//     Term 63 (AT2002-0250)/CC Outputs/Current setpoint value Ch.14 <-> Data Pointer/CurrentSetpointValues[13]
//     Term 63 (AT2002-0250)/CC Outputs/Current setpoint value Ch.15 <-> Data Pointer/CurrentSetpointValues[14]
//     Term 63 (AT2002-0250)/CC Outputs/Current setpoint value Ch.2 <-> Data Pointer/CurrentSetpointValues[1]
//     Term 63 (AT2002-0250)/CC Outputs/Current setpoint value Ch.3 <-> Data Pointer/CurrentSetpointValues[2]
//     Term 63 (AT2002-0250)/CC Outputs/Current setpoint value Ch.4 <-> Data Pointer/CurrentSetpointValues[3]
//     Term 63 (AT2002-0250)/CC Outputs/Current setpoint value Ch.5 <-> Data Pointer/CurrentSetpointValues[4]
//     Term 63 (AT2002-0250)/CC Outputs/Current setpoint value Ch.6 <-> Data Pointer/CurrentSetpointValues[5]
//     Term 63 (AT2002-0250)/CC Outputs/Current setpoint value Ch.7 <-> Data Pointer/CurrentSetpointValues[6]
//     Term 63 (AT2002-0250)/CC Outputs/Current setpoint value Ch.8 <-> Data Pointer/CurrentSetpointValues[7]
//     Term 63 (AT2002-0250)/CC Outputs/Current setpoint value Ch.9 <-> Data Pointer/CurrentSetpointValues[8]
//     Term 63 (AT2002-0250)/Term 64 (AT2002-5250)/FB Inputs/Value Channel 01 <-> Data Pointer/RawPositionValues[0]
//     Term 63 (AT2002-0250)/Term 64 (AT2002-5250)/FB Inputs/Value Channel 02 <-> Data Pointer/RawPositionValues[1]
//     Term 63 (AT2002-0250)/Term 64 (AT2002-5250)/FB Inputs/Value Channel 03 <-> Data Pointer/RawPositionValues[2]
//     Term 63 (AT2002-0250)/Term 64 (AT2002-5250)/FB Inputs/Value Channel 04 <-> Data Pointer/RawPositionValues[3]
//     Term 63 (AT2002-0250)/Term 64 (AT2002-5250)/FB Inputs/Value Channel 05 <-> Data Pointer/RawPositionValues[4]
//     Term 63 (AT2002-0250)/Term 64 (AT2002-5250)/FB Inputs/Value Channel 06 <-> Data Pointer/RawPositionValues[5]
//     Term 63 (AT2002-0250)/Term 64 (AT2002-5250)/FB Inputs/Value Channel 07 <-> Data Pointer/RawPositionValues[6]
//     Term 63 (AT2002-0250)/Term 64 (AT2002-5250)/FB Inputs/Value Channel 08 <-> Data Pointer/RawPositionValues[7]
//     Term 63 (AT2002-0250)/Term 64 (AT2002-5250)/FB Inputs/Value Channel 09 <-> Data Pointer/RawPositionValues[8]
//     Term 63 (AT2002-0250)/Term 64 (AT2002-5250)/FB Inputs/Value Channel 10 <-> Data Pointer/RawPositionValues[9]
//     Term 63 (AT2002-0250)/Term 64 (AT2002-5250)/FB Inputs/Value Channel 11 <-> Data Pointer/RawPositionValues[10]
//     Term 63 (AT2002-0250)/Term 64 (AT2002-5250)/FB Inputs/Value Channel 12 <-> Data Pointer/RawPositionValues[11]
//     Term 63 (AT2002-0250)/Term 64 (AT2002-5250)/FB Inputs/Value Channel 13 <-> Data Pointer/RawPositionValues[12]
//     Term 63 (AT2002-0250)/Term 64 (AT2002-5250)/FB Inputs/Value Channel 14 <-> Data Pointer/RawPositionValues[13]
//     Term 63 (AT2002-0250)/Term 64 (AT2002-5250)/FB Inputs/Value Channel 15 <-> Data Pointer/RawPositionValues[14]
//     Term 63 (AT2002-0250)/Term 64 (AT2002-5250)/FB Inputs/Value Channel 16 <-> Data Pointer/RawPositionValues[15]
//     Term 63 (AT2002-0250)/Term 64 (AT2002-5250)/FB Inputs/Value Channel 17 <-> Data Pointer/RawPositionValues[16]
//     Term 63 (AT2002-0250)/Term 64 (AT2002-5250)/FB Inputs/Value Channel 18 <-> Data Pointer/RawPositionValues[17]
//     Term 63 (AT2002-0250)/Term 64 (AT2002-5250)/FB Inputs/Value Channel 19 <-> Data Pointer/RawPositionValues[18]
//     Term 63 (AT2002-0250)/Term 64 (AT2002-5250)/FB Inputs/Value Channel 20 <-> Data Pointer/RawPositionValues[19]
//     Term 63 (AT2002-0250)/Term 64 (AT2002-5250)/FB Inputs/Value Channel 21 <-> Data Pointer/RawPositionValues[20]
//     Term 63 (AT2002-0250)/Term 64 (AT2002-5250)/FB Inputs/Value Channel 22 <-> Data Pointer/RawPositionValues[21]
//     Term 63 (AT2002-0250)/Term 64 (AT2002-5250)/FB Inputs/Value Channel 23 <-> Data Pointer/RawPositionValues[22]
//     Term 63 (AT2002-0250)/Term 64 (AT2002-5250)/FB Inputs/Value Channel 24 <-> Data Pointer/RawPositionValues[23]
//     Term 63 (AT2002-0250)/Term 64 (AT2002-5250)/FB Inputs/Value Channel 25 <-> Data Pointer/RawPositionValues[24]
//     Term 63 (AT2002-0250)/Term 64 (AT2002-5250)/FB Inputs/Value Channel 26 <-> Data Pointer/RawPositionValues[25]
//     Term 63 (AT2002-0250)/Term 64 (AT2002-5250)/FB Inputs/Value Channel 27 <-> Data Pointer/RawPositionValues[26]
//     Term 63 (AT2002-0250)/Term 64 (AT2002-5250)/FB Inputs/Value Channel 28 <-> Data Pointer/RawPositionValues[27]
//     Term 63 (AT2002-0250)/Term 64 (AT2002-5250)/FB Inputs/Value Channel 29 <-> Data Pointer/RawPositionValues[28]
//     Term 63 (AT2002-0250)/Term 64 (AT2002-5250)/FB Inputs/Value Channel 30 <-> Data Pointer/RawPositionValues[29]
//     Term 63 (AT2002-0250)/Term 64 (AT2002-5250)/FB Inputs/Value Channel 31 <-> Data Pointer/RawPositionValues[30]
//     Term 63 (AT2002-0250)/Term 64 (AT2002-5250)/FB Inputs/Value Channel 32 <-> Data Pointer/RawPositionValues[31]
//   Device 9 <-> TcCOM Objects/XTS ProcessingUnit 1/Part 1/Module 33
//     Term 65 (AT2000-0250)/CC Inputs/Current actual value Ch.1 <-> Data Pointer/CurrentActualValues[0]
//     Term 65 (AT2000-0250)/CC Inputs/Current actual value Ch.10 <-> Data Pointer/CurrentActualValues[9]
//     Term 65 (AT2000-0250)/CC Inputs/Current actual value Ch.11 <-> Data Pointer/CurrentActualValues[10]
//     Term 65 (AT2000-0250)/CC Inputs/Current actual value Ch.12 <-> Data Pointer/CurrentActualValues[11]
//     Term 65 (AT2000-0250)/CC Inputs/Current actual value Ch.13 <-> Data Pointer/CurrentActualValues[12]
//     Term 65 (AT2000-0250)/CC Inputs/Current actual value Ch.14 <-> Data Pointer/CurrentActualValues[13]
//     Term 65 (AT2000-0250)/CC Inputs/Current actual value Ch.15 <-> Data Pointer/CurrentActualValues[14]
//     Term 65 (AT2000-0250)/CC Inputs/Current actual value Ch.2 <-> Data Pointer/CurrentActualValues[1]
//     Term 65 (AT2000-0250)/CC Inputs/Current actual value Ch.3 <-> Data Pointer/CurrentActualValues[2]
//     Term 65 (AT2000-0250)/CC Inputs/Current actual value Ch.4 <-> Data Pointer/CurrentActualValues[3]
//     Term 65 (AT2000-0250)/CC Inputs/Current actual value Ch.5 <-> Data Pointer/CurrentActualValues[4]
//     Term 65 (AT2000-0250)/CC Inputs/Current actual value Ch.6 <-> Data Pointer/CurrentActualValues[5]
//     Term 65 (AT2000-0250)/CC Inputs/Current actual value Ch.7 <-> Data Pointer/CurrentActualValues[6]
//     Term 65 (AT2000-0250)/CC Inputs/Current actual value Ch.8 <-> Data Pointer/CurrentActualValues[7]
//     Term 65 (AT2000-0250)/CC Inputs/Current actual value Ch.9 <-> Data Pointer/CurrentActualValues[8]
//     Term 65 (AT2000-0250)/CC Inputs/Status <-> Data Pointer/Status
//     Term 65 (AT2000-0250)/CC Outputs/Control <-> Data Pointer/Control
//     Term 65 (AT2000-0250)/CC Outputs/Current setpoint value Ch.1 <-> Data Pointer/CurrentSetpointValues[0]
//     Term 65 (AT2000-0250)/CC Outputs/Current setpoint value Ch.10 <-> Data Pointer/CurrentSetpointValues[9]
//     Term 65 (AT2000-0250)/CC Outputs/Current setpoint value Ch.11 <-> Data Pointer/CurrentSetpointValues[10]
//     Term 65 (AT2000-0250)/CC Outputs/Current setpoint value Ch.12 <-> Data Pointer/CurrentSetpointValues[11]
//     Term 65 (AT2000-0250)/CC Outputs/Current setpoint value Ch.13 <-> Data Pointer/CurrentSetpointValues[12]
//     Term 65 (AT2000-0250)/CC Outputs/Current setpoint value Ch.14 <-> Data Pointer/CurrentSetpointValues[13]
//     Term 65 (AT2000-0250)/CC Outputs/Current setpoint value Ch.15 <-> Data Pointer/CurrentSetpointValues[14]
//     Term 65 (AT2000-0250)/CC Outputs/Current setpoint value Ch.2 <-> Data Pointer/CurrentSetpointValues[1]
//     Term 65 (AT2000-0250)/CC Outputs/Current setpoint value Ch.3 <-> Data Pointer/CurrentSetpointValues[2]
//     Term 65 (AT2000-0250)/CC Outputs/Current setpoint value Ch.4 <-> Data Pointer/CurrentSetpointValues[3]
//     Term 65 (AT2000-0250)/CC Outputs/Current setpoint value Ch.5 <-> Data Pointer/CurrentSetpointValues[4]
//     Term 65 (AT2000-0250)/CC Outputs/Current setpoint value Ch.6 <-> Data Pointer/CurrentSetpointValues[5]
//     Term 65 (AT2000-0250)/CC Outputs/Current setpoint value Ch.7 <-> Data Pointer/CurrentSetpointValues[6]
//     Term 65 (AT2000-0250)/CC Outputs/Current setpoint value Ch.8 <-> Data Pointer/CurrentSetpointValues[7]
//     Term 65 (AT2000-0250)/CC Outputs/Current setpoint value Ch.9 <-> Data Pointer/CurrentSetpointValues[8]
//     Term 65 (AT2000-0250)/Term 66 (AT2000-5250)/FB Inputs/Value Channel 01 <-> Data Pointer/RawPositionValues[0]
//     Term 65 (AT2000-0250)/Term 66 (AT2000-5250)/FB Inputs/Value Channel 02 <-> Data Pointer/RawPositionValues[1]
//     Term 65 (AT2000-0250)/Term 66 (AT2000-5250)/FB Inputs/Value Channel 03 <-> Data Pointer/RawPositionValues[2]
//     Term 65 (AT2000-0250)/Term 66 (AT2000-5250)/FB Inputs/Value Channel 04 <-> Data Pointer/RawPositionValues[3]
//     Term 65 (AT2000-0250)/Term 66 (AT2000-5250)/FB Inputs/Value Channel 05 <-> Data Pointer/RawPositionValues[4]
//     Term 65 (AT2000-0250)/Term 66 (AT2000-5250)/FB Inputs/Value Channel 06 <-> Data Pointer/RawPositionValues[5]
//     Term 65 (AT2000-0250)/Term 66 (AT2000-5250)/FB Inputs/Value Channel 07 <-> Data Pointer/RawPositionValues[6]
//     Term 65 (AT2000-0250)/Term 66 (AT2000-5250)/FB Inputs/Value Channel 08 <-> Data Pointer/RawPositionValues[7]
//     Term 65 (AT2000-0250)/Term 66 (AT2000-5250)/FB Inputs/Value Channel 09 <-> Data Pointer/RawPositionValues[8]
//     Term 65 (AT2000-0250)/Term 66 (AT2000-5250)/FB Inputs/Value Channel 10 <-> Data Pointer/RawPositionValues[9]
//     Term 65 (AT2000-0250)/Term 66 (AT2000-5250)/FB Inputs/Value Channel 11 <-> Data Pointer/RawPositionValues[10]
//     Term 65 (AT2000-0250)/Term 66 (AT2000-5250)/FB Inputs/Value Channel 12 <-> Data Pointer/RawPositionValues[11]
//     Term 65 (AT2000-0250)/Term 66 (AT2000-5250)/FB Inputs/Value Channel 13 <-> Data Pointer/RawPositionValues[12]
//     Term 65 (AT2000-0250)/Term 66 (AT2000-5250)/FB Inputs/Value Channel 14 <-> Data Pointer/RawPositionValues[13]
//     Term 65 (AT2000-0250)/Term 66 (AT2000-5250)/FB Inputs/Value Channel 15 <-> Data Pointer/RawPositionValues[14]
//     Term 65 (AT2000-0250)/Term 66 (AT2000-5250)/FB Inputs/Value Channel 16 <-> Data Pointer/RawPositionValues[15]
//     Term 65 (AT2000-0250)/Term 66 (AT2000-5250)/FB Inputs/Value Channel 17 <-> Data Pointer/RawPositionValues[16]
//     Term 65 (AT2000-0250)/Term 66 (AT2000-5250)/FB Inputs/Value Channel 18 <-> Data Pointer/RawPositionValues[17]
//     Term 65 (AT2000-0250)/Term 66 (AT2000-5250)/FB Inputs/Value Channel 19 <-> Data Pointer/RawPositionValues[18]
//     Term 65 (AT2000-0250)/Term 66 (AT2000-5250)/FB Inputs/Value Channel 20 <-> Data Pointer/RawPositionValues[19]
//     Term 65 (AT2000-0250)/Term 66 (AT2000-5250)/FB Inputs/Value Channel 21 <-> Data Pointer/RawPositionValues[20]
//     Term 65 (AT2000-0250)/Term 66 (AT2000-5250)/FB Inputs/Value Channel 22 <-> Data Pointer/RawPositionValues[21]
//     Term 65 (AT2000-0250)/Term 66 (AT2000-5250)/FB Inputs/Value Channel 23 <-> Data Pointer/RawPositionValues[22]
//     Term 65 (AT2000-0250)/Term 66 (AT2000-5250)/FB Inputs/Value Channel 24 <-> Data Pointer/RawPositionValues[23]
//     Term 65 (AT2000-0250)/Term 66 (AT2000-5250)/FB Inputs/Value Channel 25 <-> Data Pointer/RawPositionValues[24]
//     Term 65 (AT2000-0250)/Term 66 (AT2000-5250)/FB Inputs/Value Channel 26 <-> Data Pointer/RawPositionValues[25]
//     Term 65 (AT2000-0250)/Term 66 (AT2000-5250)/FB Inputs/Value Channel 27 <-> Data Pointer/RawPositionValues[26]
//     Term 65 (AT2000-0250)/Term 66 (AT2000-5250)/FB Inputs/Value Channel 28 <-> Data Pointer/RawPositionValues[27]
//     Term 65 (AT2000-0250)/Term 66 (AT2000-5250)/FB Inputs/Value Channel 29 <-> Data Pointer/RawPositionValues[28]
//     Term 65 (AT2000-0250)/Term 66 (AT2000-5250)/FB Inputs/Value Channel 30 <-> Data Pointer/RawPositionValues[29]
//     Term 65 (AT2000-0250)/Term 66 (AT2000-5250)/FB Inputs/Value Channel 31 <-> Data Pointer/RawPositionValues[30]
//     Term 65 (AT2000-0250)/Term 66 (AT2000-5250)/FB Inputs/Value Channel 32 <-> Data Pointer/RawPositionValues[31]
//   Device 9 <-> TcCOM Objects/XTS ProcessingUnit 1/Part 1/Module 34
//     Term 67 (AT2000-0250)/CC Inputs/Current actual value Ch.1 <-> Data Pointer/CurrentActualValues[0]
//     Term 67 (AT2000-0250)/CC Inputs/Current actual value Ch.10 <-> Data Pointer/CurrentActualValues[9]
//     Term 67 (AT2000-0250)/CC Inputs/Current actual value Ch.11 <-> Data Pointer/CurrentActualValues[10]
//     Term 67 (AT2000-0250)/CC Inputs/Current actual value Ch.12 <-> Data Pointer/CurrentActualValues[11]
//     Term 67 (AT2000-0250)/CC Inputs/Current actual value Ch.13 <-> Data Pointer/CurrentActualValues[12]
//     Term 67 (AT2000-0250)/CC Inputs/Current actual value Ch.14 <-> Data Pointer/CurrentActualValues[13]
//     Term 67 (AT2000-0250)/CC Inputs/Current actual value Ch.15 <-> Data Pointer/CurrentActualValues[14]
//     Term 67 (AT2000-0250)/CC Inputs/Current actual value Ch.2 <-> Data Pointer/CurrentActualValues[1]
//     Term 67 (AT2000-0250)/CC Inputs/Current actual value Ch.3 <-> Data Pointer/CurrentActualValues[2]
//     Term 67 (AT2000-0250)/CC Inputs/Current actual value Ch.4 <-> Data Pointer/CurrentActualValues[3]
//     Term 67 (AT2000-0250)/CC Inputs/Current actual value Ch.5 <-> Data Pointer/CurrentActualValues[4]
//     Term 67 (AT2000-0250)/CC Inputs/Current actual value Ch.6 <-> Data Pointer/CurrentActualValues[5]
//     Term 67 (AT2000-0250)/CC Inputs/Current actual value Ch.7 <-> Data Pointer/CurrentActualValues[6]
//     Term 67 (AT2000-0250)/CC Inputs/Current actual value Ch.8 <-> Data Pointer/CurrentActualValues[7]
//     Term 67 (AT2000-0250)/CC Inputs/Current actual value Ch.9 <-> Data Pointer/CurrentActualValues[8]
//     Term 67 (AT2000-0250)/CC Inputs/Status <-> Data Pointer/Status
//     Term 67 (AT2000-0250)/CC Outputs/Control <-> Data Pointer/Control
//     Term 67 (AT2000-0250)/CC Outputs/Current setpoint value Ch.1 <-> Data Pointer/CurrentSetpointValues[0]
//     Term 67 (AT2000-0250)/CC Outputs/Current setpoint value Ch.10 <-> Data Pointer/CurrentSetpointValues[9]
//     Term 67 (AT2000-0250)/CC Outputs/Current setpoint value Ch.11 <-> Data Pointer/CurrentSetpointValues[10]
//     Term 67 (AT2000-0250)/CC Outputs/Current setpoint value Ch.12 <-> Data Pointer/CurrentSetpointValues[11]
//     Term 67 (AT2000-0250)/CC Outputs/Current setpoint value Ch.13 <-> Data Pointer/CurrentSetpointValues[12]
//     Term 67 (AT2000-0250)/CC Outputs/Current setpoint value Ch.14 <-> Data Pointer/CurrentSetpointValues[13]
//     Term 67 (AT2000-0250)/CC Outputs/Current setpoint value Ch.15 <-> Data Pointer/CurrentSetpointValues[14]
//     Term 67 (AT2000-0250)/CC Outputs/Current setpoint value Ch.2 <-> Data Pointer/CurrentSetpointValues[1]
//     Term 67 (AT2000-0250)/CC Outputs/Current setpoint value Ch.3 <-> Data Pointer/CurrentSetpointValues[2]
//     Term 67 (AT2000-0250)/CC Outputs/Current setpoint value Ch.4 <-> Data Pointer/CurrentSetpointValues[3]
//     Term 67 (AT2000-0250)/CC Outputs/Current setpoint value Ch.5 <-> Data Pointer/CurrentSetpointValues[4]
//     Term 67 (AT2000-0250)/CC Outputs/Current setpoint value Ch.6 <-> Data Pointer/CurrentSetpointValues[5]
//     Term 67 (AT2000-0250)/CC Outputs/Current setpoint value Ch.7 <-> Data Pointer/CurrentSetpointValues[6]
//     Term 67 (AT2000-0250)/CC Outputs/Current setpoint value Ch.8 <-> Data Pointer/CurrentSetpointValues[7]
//     Term 67 (AT2000-0250)/CC Outputs/Current setpoint value Ch.9 <-> Data Pointer/CurrentSetpointValues[8]
//     Term 67 (AT2000-0250)/Term 68 (AT2000-5250)/FB Inputs/Value Channel 01 <-> Data Pointer/RawPositionValues[0]
//     Term 67 (AT2000-0250)/Term 68 (AT2000-5250)/FB Inputs/Value Channel 02 <-> Data Pointer/RawPositionValues[1]
//     Term 67 (AT2000-0250)/Term 68 (AT2000-5250)/FB Inputs/Value Channel 03 <-> Data Pointer/RawPositionValues[2]
//     Term 67 (AT2000-0250)/Term 68 (AT2000-5250)/FB Inputs/Value Channel 04 <-> Data Pointer/RawPositionValues[3]
//     Term 67 (AT2000-0250)/Term 68 (AT2000-5250)/FB Inputs/Value Channel 05 <-> Data Pointer/RawPositionValues[4]
//     Term 67 (AT2000-0250)/Term 68 (AT2000-5250)/FB Inputs/Value Channel 06 <-> Data Pointer/RawPositionValues[5]
//     Term 67 (AT2000-0250)/Term 68 (AT2000-5250)/FB Inputs/Value Channel 07 <-> Data Pointer/RawPositionValues[6]
//     Term 67 (AT2000-0250)/Term 68 (AT2000-5250)/FB Inputs/Value Channel 08 <-> Data Pointer/RawPositionValues[7]
//     Term 67 (AT2000-0250)/Term 68 (AT2000-5250)/FB Inputs/Value Channel 09 <-> Data Pointer/RawPositionValues[8]
//     Term 67 (AT2000-0250)/Term 68 (AT2000-5250)/FB Inputs/Value Channel 10 <-> Data Pointer/RawPositionValues[9]
//     Term 67 (AT2000-0250)/Term 68 (AT2000-5250)/FB Inputs/Value Channel 11 <-> Data Pointer/RawPositionValues[10]
//     Term 67 (AT2000-0250)/Term 68 (AT2000-5250)/FB Inputs/Value Channel 12 <-> Data Pointer/RawPositionValues[11]
//     Term 67 (AT2000-0250)/Term 68 (AT2000-5250)/FB Inputs/Value Channel 13 <-> Data Pointer/RawPositionValues[12]
//     Term 67 (AT2000-0250)/Term 68 (AT2000-5250)/FB Inputs/Value Channel 14 <-> Data Pointer/RawPositionValues[13]
//     Term 67 (AT2000-0250)/Term 68 (AT2000-5250)/FB Inputs/Value Channel 15 <-> Data Pointer/RawPositionValues[14]
//     Term 67 (AT2000-0250)/Term 68 (AT2000-5250)/FB Inputs/Value Channel 16 <-> Data Pointer/RawPositionValues[15]
//     Term 67 (AT2000-0250)/Term 68 (AT2000-5250)/FB Inputs/Value Channel 17 <-> Data Pointer/RawPositionValues[16]
//     Term 67 (AT2000-0250)/Term 68 (AT2000-5250)/FB Inputs/Value Channel 18 <-> Data Pointer/RawPositionValues[17]
//     Term 67 (AT2000-0250)/Term 68 (AT2000-5250)/FB Inputs/Value Channel 19 <-> Data Pointer/RawPositionValues[18]
//     Term 67 (AT2000-0250)/Term 68 (AT2000-5250)/FB Inputs/Value Channel 20 <-> Data Pointer/RawPositionValues[19]
//     Term 67 (AT2000-0250)/Term 68 (AT2000-5250)/FB Inputs/Value Channel 21 <-> Data Pointer/RawPositionValues[20]
//     Term 67 (AT2000-0250)/Term 68 (AT2000-5250)/FB Inputs/Value Channel 22 <-> Data Pointer/RawPositionValues[21]
//     Term 67 (AT2000-0250)/Term 68 (AT2000-5250)/FB Inputs/Value Channel 23 <-> Data Pointer/RawPositionValues[22]
//     Term 67 (AT2000-0250)/Term 68 (AT2000-5250)/FB Inputs/Value Channel 24 <-> Data Pointer/RawPositionValues[23]
//     Term 67 (AT2000-0250)/Term 68 (AT2000-5250)/FB Inputs/Value Channel 25 <-> Data Pointer/RawPositionValues[24]
//     Term 67 (AT2000-0250)/Term 68 (AT2000-5250)/FB Inputs/Value Channel 26 <-> Data Pointer/RawPositionValues[25]
//     Term 67 (AT2000-0250)/Term 68 (AT2000-5250)/FB Inputs/Value Channel 27 <-> Data Pointer/RawPositionValues[26]
//     Term 67 (AT2000-0250)/Term 68 (AT2000-5250)/FB Inputs/Value Channel 28 <-> Data Pointer/RawPositionValues[27]
//     Term 67 (AT2000-0250)/Term 68 (AT2000-5250)/FB Inputs/Value Channel 29 <-> Data Pointer/RawPositionValues[28]
//     Term 67 (AT2000-0250)/Term 68 (AT2000-5250)/FB Inputs/Value Channel 30 <-> Data Pointer/RawPositionValues[29]
//     Term 67 (AT2000-0250)/Term 68 (AT2000-5250)/FB Inputs/Value Channel 31 <-> Data Pointer/RawPositionValues[30]
//     Term 67 (AT2000-0250)/Term 68 (AT2000-5250)/FB Inputs/Value Channel 32 <-> Data Pointer/RawPositionValues[31]
//   Device 9 <-> TcCOM Objects/XTS ProcessingUnit 1/Part 1/Module 35
//     Term 69 (AT2000-0250)/CC Inputs/Current actual value Ch.1 <-> Data Pointer/CurrentActualValues[0]
//     Term 69 (AT2000-0250)/CC Inputs/Current actual value Ch.10 <-> Data Pointer/CurrentActualValues[9]
//     Term 69 (AT2000-0250)/CC Inputs/Current actual value Ch.11 <-> Data Pointer/CurrentActualValues[10]
//     Term 69 (AT2000-0250)/CC Inputs/Current actual value Ch.12 <-> Data Pointer/CurrentActualValues[11]
//     Term 69 (AT2000-0250)/CC Inputs/Current actual value Ch.13 <-> Data Pointer/CurrentActualValues[12]
//     Term 69 (AT2000-0250)/CC Inputs/Current actual value Ch.14 <-> Data Pointer/CurrentActualValues[13]
//     Term 69 (AT2000-0250)/CC Inputs/Current actual value Ch.15 <-> Data Pointer/CurrentActualValues[14]
//     Term 69 (AT2000-0250)/CC Inputs/Current actual value Ch.2 <-> Data Pointer/CurrentActualValues[1]
//     Term 69 (AT2000-0250)/CC Inputs/Current actual value Ch.3 <-> Data Pointer/CurrentActualValues[2]
//     Term 69 (AT2000-0250)/CC Inputs/Current actual value Ch.4 <-> Data Pointer/CurrentActualValues[3]
//     Term 69 (AT2000-0250)/CC Inputs/Current actual value Ch.5 <-> Data Pointer/CurrentActualValues[4]
//     Term 69 (AT2000-0250)/CC Inputs/Current actual value Ch.6 <-> Data Pointer/CurrentActualValues[5]
//     Term 69 (AT2000-0250)/CC Inputs/Current actual value Ch.7 <-> Data Pointer/CurrentActualValues[6]
//     Term 69 (AT2000-0250)/CC Inputs/Current actual value Ch.8 <-> Data Pointer/CurrentActualValues[7]
//     Term 69 (AT2000-0250)/CC Inputs/Current actual value Ch.9 <-> Data Pointer/CurrentActualValues[8]
//     Term 69 (AT2000-0250)/CC Inputs/Status <-> Data Pointer/Status
//     Term 69 (AT2000-0250)/CC Outputs/Control <-> Data Pointer/Control
//     Term 69 (AT2000-0250)/CC Outputs/Current setpoint value Ch.1 <-> Data Pointer/CurrentSetpointValues[0]
//     Term 69 (AT2000-0250)/CC Outputs/Current setpoint value Ch.10 <-> Data Pointer/CurrentSetpointValues[9]
//     Term 69 (AT2000-0250)/CC Outputs/Current setpoint value Ch.11 <-> Data Pointer/CurrentSetpointValues[10]
//     Term 69 (AT2000-0250)/CC Outputs/Current setpoint value Ch.12 <-> Data Pointer/CurrentSetpointValues[11]
//     Term 69 (AT2000-0250)/CC Outputs/Current setpoint value Ch.13 <-> Data Pointer/CurrentSetpointValues[12]
//     Term 69 (AT2000-0250)/CC Outputs/Current setpoint value Ch.14 <-> Data Pointer/CurrentSetpointValues[13]
//     Term 69 (AT2000-0250)/CC Outputs/Current setpoint value Ch.15 <-> Data Pointer/CurrentSetpointValues[14]
//     Term 69 (AT2000-0250)/CC Outputs/Current setpoint value Ch.2 <-> Data Pointer/CurrentSetpointValues[1]
//     Term 69 (AT2000-0250)/CC Outputs/Current setpoint value Ch.3 <-> Data Pointer/CurrentSetpointValues[2]
//     Term 69 (AT2000-0250)/CC Outputs/Current setpoint value Ch.4 <-> Data Pointer/CurrentSetpointValues[3]
//     Term 69 (AT2000-0250)/CC Outputs/Current setpoint value Ch.5 <-> Data Pointer/CurrentSetpointValues[4]
//     Term 69 (AT2000-0250)/CC Outputs/Current setpoint value Ch.6 <-> Data Pointer/CurrentSetpointValues[5]
//     Term 69 (AT2000-0250)/CC Outputs/Current setpoint value Ch.7 <-> Data Pointer/CurrentSetpointValues[6]
//     Term 69 (AT2000-0250)/CC Outputs/Current setpoint value Ch.8 <-> Data Pointer/CurrentSetpointValues[7]
//     Term 69 (AT2000-0250)/CC Outputs/Current setpoint value Ch.9 <-> Data Pointer/CurrentSetpointValues[8]
//     Term 69 (AT2000-0250)/Term 70 (AT2000-5250)/FB Inputs/Value Channel 01 <-> Data Pointer/RawPositionValues[0]
//     Term 69 (AT2000-0250)/Term 70 (AT2000-5250)/FB Inputs/Value Channel 02 <-> Data Pointer/RawPositionValues[1]
//     Term 69 (AT2000-0250)/Term 70 (AT2000-5250)/FB Inputs/Value Channel 03 <-> Data Pointer/RawPositionValues[2]
//     Term 69 (AT2000-0250)/Term 70 (AT2000-5250)/FB Inputs/Value Channel 04 <-> Data Pointer/RawPositionValues[3]
//     Term 69 (AT2000-0250)/Term 70 (AT2000-5250)/FB Inputs/Value Channel 05 <-> Data Pointer/RawPositionValues[4]
//     Term 69 (AT2000-0250)/Term 70 (AT2000-5250)/FB Inputs/Value Channel 06 <-> Data Pointer/RawPositionValues[5]
//     Term 69 (AT2000-0250)/Term 70 (AT2000-5250)/FB Inputs/Value Channel 07 <-> Data Pointer/RawPositionValues[6]
//     Term 69 (AT2000-0250)/Term 70 (AT2000-5250)/FB Inputs/Value Channel 08 <-> Data Pointer/RawPositionValues[7]
//     Term 69 (AT2000-0250)/Term 70 (AT2000-5250)/FB Inputs/Value Channel 09 <-> Data Pointer/RawPositionValues[8]
//     Term 69 (AT2000-0250)/Term 70 (AT2000-5250)/FB Inputs/Value Channel 10 <-> Data Pointer/RawPositionValues[9]
//     Term 69 (AT2000-0250)/Term 70 (AT2000-5250)/FB Inputs/Value Channel 11 <-> Data Pointer/RawPositionValues[10]
//     Term 69 (AT2000-0250)/Term 70 (AT2000-5250)/FB Inputs/Value Channel 12 <-> Data Pointer/RawPositionValues[11]
//     Term 69 (AT2000-0250)/Term 70 (AT2000-5250)/FB Inputs/Value Channel 13 <-> Data Pointer/RawPositionValues[12]
//     Term 69 (AT2000-0250)/Term 70 (AT2000-5250)/FB Inputs/Value Channel 14 <-> Data Pointer/RawPositionValues[13]
//     Term 69 (AT2000-0250)/Term 70 (AT2000-5250)/FB Inputs/Value Channel 15 <-> Data Pointer/RawPositionValues[14]
//     Term 69 (AT2000-0250)/Term 70 (AT2000-5250)/FB Inputs/Value Channel 16 <-> Data Pointer/RawPositionValues[15]
//     Term 69 (AT2000-0250)/Term 70 (AT2000-5250)/FB Inputs/Value Channel 17 <-> Data Pointer/RawPositionValues[16]
//     Term 69 (AT2000-0250)/Term 70 (AT2000-5250)/FB Inputs/Value Channel 18 <-> Data Pointer/RawPositionValues[17]
//     Term 69 (AT2000-0250)/Term 70 (AT2000-5250)/FB Inputs/Value Channel 19 <-> Data Pointer/RawPositionValues[18]
//     Term 69 (AT2000-0250)/Term 70 (AT2000-5250)/FB Inputs/Value Channel 20 <-> Data Pointer/RawPositionValues[19]
//     Term 69 (AT2000-0250)/Term 70 (AT2000-5250)/FB Inputs/Value Channel 21 <-> Data Pointer/RawPositionValues[20]
//     Term 69 (AT2000-0250)/Term 70 (AT2000-5250)/FB Inputs/Value Channel 22 <-> Data Pointer/RawPositionValues[21]
//     Term 69 (AT2000-0250)/Term 70 (AT2000-5250)/FB Inputs/Value Channel 23 <-> Data Pointer/RawPositionValues[22]
//     Term 69 (AT2000-0250)/Term 70 (AT2000-5250)/FB Inputs/Value Channel 24 <-> Data Pointer/RawPositionValues[23]
//     Term 69 (AT2000-0250)/Term 70 (AT2000-5250)/FB Inputs/Value Channel 25 <-> Data Pointer/RawPositionValues[24]
//     Term 69 (AT2000-0250)/Term 70 (AT2000-5250)/FB Inputs/Value Channel 26 <-> Data Pointer/RawPositionValues[25]
//     Term 69 (AT2000-0250)/Term 70 (AT2000-5250)/FB Inputs/Value Channel 27 <-> Data Pointer/RawPositionValues[26]
//     Term 69 (AT2000-0250)/Term 70 (AT2000-5250)/FB Inputs/Value Channel 28 <-> Data Pointer/RawPositionValues[27]
//     Term 69 (AT2000-0250)/Term 70 (AT2000-5250)/FB Inputs/Value Channel 29 <-> Data Pointer/RawPositionValues[28]
//     Term 69 (AT2000-0250)/Term 70 (AT2000-5250)/FB Inputs/Value Channel 30 <-> Data Pointer/RawPositionValues[29]
//     Term 69 (AT2000-0250)/Term 70 (AT2000-5250)/FB Inputs/Value Channel 31 <-> Data Pointer/RawPositionValues[30]
//     Term 69 (AT2000-0250)/Term 70 (AT2000-5250)/FB Inputs/Value Channel 32 <-> Data Pointer/RawPositionValues[31]
//   ExternControl/ExternControl Instance <-> XtsTransport/XtsTransport Instance
//     PLC_1 Inputs/MAPPING_in.AppState.byState <-> PLC_1 Outputs/MAPPING_out.AppState.byState
//     PLC_1 Inputs/MAPPING_in.InstanceState.byState <-> PLC_1 Outputs/MAPPING_out.InstanceState.byState
//     PLC_1 Inputs/MAPPING_in.TicketListOutput.byData <-> PLC_1 Outputs/MAPPING_out.TicketListOutput.byData
//     PLC_1 Inputs/MAPPING_in.TicketListState.byState <-> PLC_1 Outputs/MAPPING_out.TicketListState.byState
//     PLC_1 Inputs/MAPPING_in.TransportState.byState <-> PLC_1 Outputs/MAPPING_out.TransportState.byState
//     PLC_1 Outputs/MAPPING_out.AppControl.byCtrl <-> PLC_1 Inputs/MAPPING_in.AppControl.byCtrl
//     PLC_1 Outputs/MAPPING_out.InstanceCtrl.byCtrl <-> PLC_1 Inputs/MAPPING_in.InstanceControl.byCtrl
//     PLC_1 Outputs/MAPPING_out.TicketListControl.byCtrl <-> PLC_1 Inputs/MAPPING_in.TicketListControl.byCtrl
//     PLC_1 Outputs/MAPPING_out.TicketListInput.byData <-> PLC_1 Inputs/MAPPING_in.TicketListInput.byData
//     PLC_1 Outputs/MAPPING_out.TransportControl.byCtrl <-> PLC_1 Inputs/MAPPING_in.TransportControl.byCtrl
//   XtsTransport/XtsTransport Instance <-> NC-Task 1/Axes/Mover Axis 1
//     PLC_1 Inputs/GVL_XTS.AxisRefMover[1].NcToPlc <-> Outputs/ToPlc
//     PLC_1 Outputs/GVL_XTS.AxisRefMover[1].PlcToNc <-> Inputs/FromPlc
//   XtsTransport/XtsTransport Instance <-> NC-Task 1/Axes/Mover Axis 10
//     PLC_1 Inputs/GVL_XTS.AxisRefMover[10].NcToPlc <-> Outputs/ToPlc
//     PLC_1 Outputs/GVL_XTS.AxisRefMover[10].PlcToNc <-> Inputs/FromPlc
//   XtsTransport/XtsTransport Instance <-> NC-Task 1/Axes/Mover Axis 100
//     PLC_1 Inputs/GVL_XTS.AxisRefMover[100].NcToPlc <-> Outputs/ToPlc
//     PLC_1 Outputs/GVL_XTS.AxisRefMover[100].PlcToNc <-> Inputs/FromPlc
//   XtsTransport/XtsTransport Instance <-> NC-Task 1/Axes/Mover Axis 101
//     PLC_1 Inputs/GVL_XTS.AxisRefMover[101].NcToPlc <-> Outputs/ToPlc
//     PLC_1 Outputs/GVL_XTS.AxisRefMover[101].PlcToNc <-> Inputs/FromPlc
//   XtsTransport/XtsTransport Instance <-> NC-Task 1/Axes/Mover Axis 102
//     PLC_1 Inputs/GVL_XTS.AxisRefMover[102].NcToPlc <-> Outputs/ToPlc
//     PLC_1 Outputs/GVL_XTS.AxisRefMover[102].PlcToNc <-> Inputs/FromPlc
//   XtsTransport/XtsTransport Instance <-> NC-Task 1/Axes/Mover Axis 103
//     PLC_1 Inputs/GVL_XTS.AxisRefMover[103].NcToPlc <-> Outputs/ToPlc
//     PLC_1 Outputs/GVL_XTS.AxisRefMover[103].PlcToNc <-> Inputs/FromPlc
//   XtsTransport/XtsTransport Instance <-> NC-Task 1/Axes/Mover Axis 104
//     PLC_1 Inputs/GVL_XTS.AxisRefMover[104].NcToPlc <-> Outputs/ToPlc
//     PLC_1 Outputs/GVL_XTS.AxisRefMover[104].PlcToNc <-> Inputs/FromPlc
//   XtsTransport/XtsTransport Instance <-> NC-Task 1/Axes/Mover Axis 105
//     PLC_1 Inputs/GVL_XTS.AxisRefMover[105].NcToPlc <-> Outputs/ToPlc
//     PLC_1 Outputs/GVL_XTS.AxisRefMover[105].PlcToNc <-> Inputs/FromPlc
//   XtsTransport/XtsTransport Instance <-> NC-Task 1/Axes/Mover Axis 106
//     PLC_1 Inputs/GVL_XTS.AxisRefMover[106].NcToPlc <-> Outputs/ToPlc
//     PLC_1 Outputs/GVL_XTS.AxisRefMover[106].PlcToNc <-> Inputs/FromPlc
//   XtsTransport/XtsTransport Instance <-> NC-Task 1/Axes/Mover Axis 107
//     PLC_1 Inputs/GVL_XTS.AxisRefMover[107].NcToPlc <-> Outputs/ToPlc
//     PLC_1 Outputs/GVL_XTS.AxisRefMover[107].PlcToNc <-> Inputs/FromPlc
//   XtsTransport/XtsTransport Instance <-> NC-Task 1/Axes/Mover Axis 108
//     PLC_1 Inputs/GVL_XTS.AxisRefMover[108].NcToPlc <-> Outputs/ToPlc
//     PLC_1 Outputs/GVL_XTS.AxisRefMover[108].PlcToNc <-> Inputs/FromPlc
//   XtsTransport/XtsTransport Instance <-> NC-Task 1/Axes/Mover Axis 11
//     PLC_1 Inputs/GVL_XTS.AxisRefMover[11].NcToPlc <-> Outputs/ToPlc
//     PLC_1 Outputs/GVL_XTS.AxisRefMover[11].PlcToNc <-> Inputs/FromPlc
//   XtsTransport/XtsTransport Instance <-> NC-Task 1/Axes/Mover Axis 12
//     PLC_1 Inputs/GVL_XTS.AxisRefMover[12].NcToPlc <-> Outputs/ToPlc
//     PLC_1 Outputs/GVL_XTS.AxisRefMover[12].PlcToNc <-> Inputs/FromPlc
//   XtsTransport/XtsTransport Instance <-> NC-Task 1/Axes/Mover Axis 13
//     PLC_1 Inputs/GVL_XTS.AxisRefMover[13].NcToPlc <-> Outputs/ToPlc
//     PLC_1 Outputs/GVL_XTS.AxisRefMover[13].PlcToNc <-> Inputs/FromPlc
//   XtsTransport/XtsTransport Instance <-> NC-Task 1/Axes/Mover Axis 14
//     PLC_1 Inputs/GVL_XTS.AxisRefMover[14].NcToPlc <-> Outputs/ToPlc
//     PLC_1 Outputs/GVL_XTS.AxisRefMover[14].PlcToNc <-> Inputs/FromPlc
//   XtsTransport/XtsTransport Instance <-> NC-Task 1/Axes/Mover Axis 15
//     PLC_1 Inputs/GVL_XTS.AxisRefMover[15].NcToPlc <-> Outputs/ToPlc
//     PLC_1 Outputs/GVL_XTS.AxisRefMover[15].PlcToNc <-> Inputs/FromPlc
//   XtsTransport/XtsTransport Instance <-> NC-Task 1/Axes/Mover Axis 16
//     PLC_1 Inputs/GVL_XTS.AxisRefMover[16].NcToPlc <-> Outputs/ToPlc
//     PLC_1 Outputs/GVL_XTS.AxisRefMover[16].PlcToNc <-> Inputs/FromPlc
//   XtsTransport/XtsTransport Instance <-> NC-Task 1/Axes/Mover Axis 17
//     PLC_1 Inputs/GVL_XTS.AxisRefMover[17].NcToPlc <-> Outputs/ToPlc
//     PLC_1 Outputs/GVL_XTS.AxisRefMover[17].PlcToNc <-> Inputs/FromPlc
//   XtsTransport/XtsTransport Instance <-> NC-Task 1/Axes/Mover Axis 18
//     PLC_1 Inputs/GVL_XTS.AxisRefMover[18].NcToPlc <-> Outputs/ToPlc
//     PLC_1 Outputs/GVL_XTS.AxisRefMover[18].PlcToNc <-> Inputs/FromPlc
//   XtsTransport/XtsTransport Instance <-> NC-Task 1/Axes/Mover Axis 19
//     PLC_1 Inputs/GVL_XTS.AxisRefMover[19].NcToPlc <-> Outputs/ToPlc
//     PLC_1 Outputs/GVL_XTS.AxisRefMover[19].PlcToNc <-> Inputs/FromPlc
//   XtsTransport/XtsTransport Instance <-> NC-Task 1/Axes/Mover Axis 2
//     PLC_1 Inputs/GVL_XTS.AxisRefMover[2].NcToPlc <-> Outputs/ToPlc
//     PLC_1 Outputs/GVL_XTS.AxisRefMover[2].PlcToNc <-> Inputs/FromPlc
//   XtsTransport/XtsTransport Instance <-> NC-Task 1/Axes/Mover Axis 20
//     PLC_1 Inputs/GVL_XTS.AxisRefMover[20].NcToPlc <-> Outputs/ToPlc
//     PLC_1 Outputs/GVL_XTS.AxisRefMover[20].PlcToNc <-> Inputs/FromPlc
//   XtsTransport/XtsTransport Instance <-> NC-Task 1/Axes/Mover Axis 21
//     PLC_1 Inputs/GVL_XTS.AxisRefMover[21].NcToPlc <-> Outputs/ToPlc
//     PLC_1 Outputs/GVL_XTS.AxisRefMover[21].PlcToNc <-> Inputs/FromPlc
//   XtsTransport/XtsTransport Instance <-> NC-Task 1/Axes/Mover Axis 22
//     PLC_1 Inputs/GVL_XTS.AxisRefMover[22].NcToPlc <-> Outputs/ToPlc
//     PLC_1 Outputs/GVL_XTS.AxisRefMover[22].PlcToNc <-> Inputs/FromPlc
//   XtsTransport/XtsTransport Instance <-> NC-Task 1/Axes/Mover Axis 23
//     PLC_1 Inputs/GVL_XTS.AxisRefMover[23].NcToPlc <-> Outputs/ToPlc
//     PLC_1 Outputs/GVL_XTS.AxisRefMover[23].PlcToNc <-> Inputs/FromPlc
//   XtsTransport/XtsTransport Instance <-> NC-Task 1/Axes/Mover Axis 24
//     PLC_1 Inputs/GVL_XTS.AxisRefMover[24].NcToPlc <-> Outputs/ToPlc
//     PLC_1 Outputs/GVL_XTS.AxisRefMover[24].PlcToNc <-> Inputs/FromPlc
//   XtsTransport/XtsTransport Instance <-> NC-Task 1/Axes/Mover Axis 25
//     PLC_1 Inputs/GVL_XTS.AxisRefMover[25].NcToPlc <-> Outputs/ToPlc
//     PLC_1 Outputs/GVL_XTS.AxisRefMover[25].PlcToNc <-> Inputs/FromPlc
//   XtsTransport/XtsTransport Instance <-> NC-Task 1/Axes/Mover Axis 26
//     PLC_1 Inputs/GVL_XTS.AxisRefMover[26].NcToPlc <-> Outputs/ToPlc
//     PLC_1 Outputs/GVL_XTS.AxisRefMover[26].PlcToNc <-> Inputs/FromPlc
//   XtsTransport/XtsTransport Instance <-> NC-Task 1/Axes/Mover Axis 27
//     PLC_1 Inputs/GVL_XTS.AxisRefMover[27].NcToPlc <-> Outputs/ToPlc
//     PLC_1 Outputs/GVL_XTS.AxisRefMover[27].PlcToNc <-> Inputs/FromPlc
//   XtsTransport/XtsTransport Instance <-> NC-Task 1/Axes/Mover Axis 28
//     PLC_1 Inputs/GVL_XTS.AxisRefMover[28].NcToPlc <-> Outputs/ToPlc
//     PLC_1 Outputs/GVL_XTS.AxisRefMover[28].PlcToNc <-> Inputs/FromPlc
//   XtsTransport/XtsTransport Instance <-> NC-Task 1/Axes/Mover Axis 29
//     PLC_1 Inputs/GVL_XTS.AxisRefMover[29].NcToPlc <-> Outputs/ToPlc
//     PLC_1 Outputs/GVL_XTS.AxisRefMover[29].PlcToNc <-> Inputs/FromPlc
//   XtsTransport/XtsTransport Instance <-> NC-Task 1/Axes/Mover Axis 3
//     PLC_1 Inputs/GVL_XTS.AxisRefMover[3].NcToPlc <-> Outputs/ToPlc
//     PLC_1 Outputs/GVL_XTS.AxisRefMover[3].PlcToNc <-> Inputs/FromPlc
//   XtsTransport/XtsTransport Instance <-> NC-Task 1/Axes/Mover Axis 30
//     PLC_1 Inputs/GVL_XTS.AxisRefMover[30].NcToPlc <-> Outputs/ToPlc
//     PLC_1 Outputs/GVL_XTS.AxisRefMover[30].PlcToNc <-> Inputs/FromPlc
//   XtsTransport/XtsTransport Instance <-> NC-Task 1/Axes/Mover Axis 31
//     PLC_1 Inputs/GVL_XTS.AxisRefMover[31].NcToPlc <-> Outputs/ToPlc
//     PLC_1 Outputs/GVL_XTS.AxisRefMover[31].PlcToNc <-> Inputs/FromPlc
//   XtsTransport/XtsTransport Instance <-> NC-Task 1/Axes/Mover Axis 32
//     PLC_1 Inputs/GVL_XTS.AxisRefMover[32].NcToPlc <-> Outputs/ToPlc
//     PLC_1 Outputs/GVL_XTS.AxisRefMover[32].PlcToNc <-> Inputs/FromPlc
//   XtsTransport/XtsTransport Instance <-> NC-Task 1/Axes/Mover Axis 33
//     PLC_1 Inputs/GVL_XTS.AxisRefMover[33].NcToPlc <-> Outputs/ToPlc
//     PLC_1 Outputs/GVL_XTS.AxisRefMover[33].PlcToNc <-> Inputs/FromPlc
//   XtsTransport/XtsTransport Instance <-> NC-Task 1/Axes/Mover Axis 34
//     PLC_1 Inputs/GVL_XTS.AxisRefMover[34].NcToPlc <-> Outputs/ToPlc
//     PLC_1 Outputs/GVL_XTS.AxisRefMover[34].PlcToNc <-> Inputs/FromPlc
//   XtsTransport/XtsTransport Instance <-> NC-Task 1/Axes/Mover Axis 35
//     PLC_1 Inputs/GVL_XTS.AxisRefMover[35].NcToPlc <-> Outputs/ToPlc
//     PLC_1 Outputs/GVL_XTS.AxisRefMover[35].PlcToNc <-> Inputs/FromPlc
//   XtsTransport/XtsTransport Instance <-> NC-Task 1/Axes/Mover Axis 36
//     PLC_1 Inputs/GVL_XTS.AxisRefMover[36].NcToPlc <-> Outputs/ToPlc
//     PLC_1 Outputs/GVL_XTS.AxisRefMover[36].PlcToNc <-> Inputs/FromPlc
//   XtsTransport/XtsTransport Instance <-> NC-Task 1/Axes/Mover Axis 37
//     PLC_1 Inputs/GVL_XTS.AxisRefMover[37].NcToPlc <-> Outputs/ToPlc
//     PLC_1 Outputs/GVL_XTS.AxisRefMover[37].PlcToNc <-> Inputs/FromPlc
//   XtsTransport/XtsTransport Instance <-> NC-Task 1/Axes/Mover Axis 38
//     PLC_1 Inputs/GVL_XTS.AxisRefMover[38].NcToPlc <-> Outputs/ToPlc
//     PLC_1 Outputs/GVL_XTS.AxisRefMover[38].PlcToNc <-> Inputs/FromPlc
//   XtsTransport/XtsTransport Instance <-> NC-Task 1/Axes/Mover Axis 39
//     PLC_1 Inputs/GVL_XTS.AxisRefMover[39].NcToPlc <-> Outputs/ToPlc
//     PLC_1 Outputs/GVL_XTS.AxisRefMover[39].PlcToNc <-> Inputs/FromPlc
//   XtsTransport/XtsTransport Instance <-> NC-Task 1/Axes/Mover Axis 4
//     PLC_1 Inputs/GVL_XTS.AxisRefMover[4].NcToPlc <-> Outputs/ToPlc
//     PLC_1 Outputs/GVL_XTS.AxisRefMover[4].PlcToNc <-> Inputs/FromPlc
//   XtsTransport/XtsTransport Instance <-> NC-Task 1/Axes/Mover Axis 40
//     PLC_1 Inputs/GVL_XTS.AxisRefMover[40].NcToPlc <-> Outputs/ToPlc
//     PLC_1 Outputs/GVL_XTS.AxisRefMover[40].PlcToNc <-> Inputs/FromPlc
//   XtsTransport/XtsTransport Instance <-> NC-Task 1/Axes/Mover Axis 41
//     PLC_1 Inputs/GVL_XTS.AxisRefMover[41].NcToPlc <-> Outputs/ToPlc
//     PLC_1 Outputs/GVL_XTS.AxisRefMover[41].PlcToNc <-> Inputs/FromPlc
//   XtsTransport/XtsTransport Instance <-> NC-Task 1/Axes/Mover Axis 42
//     PLC_1 Inputs/GVL_XTS.AxisRefMover[42].NcToPlc <-> Outputs/ToPlc
//     PLC_1 Outputs/GVL_XTS.AxisRefMover[42].PlcToNc <-> Inputs/FromPlc
//   XtsTransport/XtsTransport Instance <-> NC-Task 1/Axes/Mover Axis 43
//     PLC_1 Inputs/GVL_XTS.AxisRefMover[43].NcToPlc <-> Outputs/ToPlc
//     PLC_1 Outputs/GVL_XTS.AxisRefMover[43].PlcToNc <-> Inputs/FromPlc
//   XtsTransport/XtsTransport Instance <-> NC-Task 1/Axes/Mover Axis 44
//     PLC_1 Inputs/GVL_XTS.AxisRefMover[44].NcToPlc <-> Outputs/ToPlc
//     PLC_1 Outputs/GVL_XTS.AxisRefMover[44].PlcToNc <-> Inputs/FromPlc
//   XtsTransport/XtsTransport Instance <-> NC-Task 1/Axes/Mover Axis 45
//     PLC_1 Inputs/GVL_XTS.AxisRefMover[45].NcToPlc <-> Outputs/ToPlc
//     PLC_1 Outputs/GVL_XTS.AxisRefMover[45].PlcToNc <-> Inputs/FromPlc
//   XtsTransport/XtsTransport Instance <-> NC-Task 1/Axes/Mover Axis 46
//     PLC_1 Inputs/GVL_XTS.AxisRefMover[46].NcToPlc <-> Outputs/ToPlc
//     PLC_1 Outputs/GVL_XTS.AxisRefMover[46].PlcToNc <-> Inputs/FromPlc
//   XtsTransport/XtsTransport Instance <-> NC-Task 1/Axes/Mover Axis 47
//     PLC_1 Inputs/GVL_XTS.AxisRefMover[47].NcToPlc <-> Outputs/ToPlc
//     PLC_1 Outputs/GVL_XTS.AxisRefMover[47].PlcToNc <-> Inputs/FromPlc
//   XtsTransport/XtsTransport Instance <-> NC-Task 1/Axes/Mover Axis 48
//     PLC_1 Inputs/GVL_XTS.AxisRefMover[48].NcToPlc <-> Outputs/ToPlc
//     PLC_1 Outputs/GVL_XTS.AxisRefMover[48].PlcToNc <-> Inputs/FromPlc
//   XtsTransport/XtsTransport Instance <-> NC-Task 1/Axes/Mover Axis 49
//     PLC_1 Inputs/GVL_XTS.AxisRefMover[49].NcToPlc <-> Outputs/ToPlc
//     PLC_1 Outputs/GVL_XTS.AxisRefMover[49].PlcToNc <-> Inputs/FromPlc
//   XtsTransport/XtsTransport Instance <-> NC-Task 1/Axes/Mover Axis 5
//     PLC_1 Inputs/GVL_XTS.AxisRefMover[5].NcToPlc <-> Outputs/ToPlc
//     PLC_1 Outputs/GVL_XTS.AxisRefMover[5].PlcToNc <-> Inputs/FromPlc
//   XtsTransport/XtsTransport Instance <-> NC-Task 1/Axes/Mover Axis 50
//     PLC_1 Inputs/GVL_XTS.AxisRefMover[50].NcToPlc <-> Outputs/ToPlc
//     PLC_1 Outputs/GVL_XTS.AxisRefMover[50].PlcToNc <-> Inputs/FromPlc
//   XtsTransport/XtsTransport Instance <-> NC-Task 1/Axes/Mover Axis 51
//     PLC_1 Inputs/GVL_XTS.AxisRefMover[51].NcToPlc <-> Outputs/ToPlc
//     PLC_1 Outputs/GVL_XTS.AxisRefMover[51].PlcToNc <-> Inputs/FromPlc
//   XtsTransport/XtsTransport Instance <-> NC-Task 1/Axes/Mover Axis 52
//     PLC_1 Inputs/GVL_XTS.AxisRefMover[52].NcToPlc <-> Outputs/ToPlc
//     PLC_1 Outputs/GVL_XTS.AxisRefMover[52].PlcToNc <-> Inputs/FromPlc
//   XtsTransport/XtsTransport Instance <-> NC-Task 1/Axes/Mover Axis 53
//     PLC_1 Inputs/GVL_XTS.AxisRefMover[53].NcToPlc <-> Outputs/ToPlc
//     PLC_1 Outputs/GVL_XTS.AxisRefMover[53].PlcToNc <-> Inputs/FromPlc
//   XtsTransport/XtsTransport Instance <-> NC-Task 1/Axes/Mover Axis 54
//     PLC_1 Inputs/GVL_XTS.AxisRefMover[54].NcToPlc <-> Outputs/ToPlc
//     PLC_1 Outputs/GVL_XTS.AxisRefMover[54].PlcToNc <-> Inputs/FromPlc
//   XtsTransport/XtsTransport Instance <-> NC-Task 1/Axes/Mover Axis 55
//     PLC_1 Inputs/GVL_XTS.AxisRefMover[55].NcToPlc <-> Outputs/ToPlc
//     PLC_1 Outputs/GVL_XTS.AxisRefMover[55].PlcToNc <-> Inputs/FromPlc
//   XtsTransport/XtsTransport Instance <-> NC-Task 1/Axes/Mover Axis 56
//     PLC_1 Inputs/GVL_XTS.AxisRefMover[56].NcToPlc <-> Outputs/ToPlc
//     PLC_1 Outputs/GVL_XTS.AxisRefMover[56].PlcToNc <-> Inputs/FromPlc
//   XtsTransport/XtsTransport Instance <-> NC-Task 1/Axes/Mover Axis 57
//     PLC_1 Inputs/GVL_XTS.AxisRefMover[57].NcToPlc <-> Outputs/ToPlc
//     PLC_1 Outputs/GVL_XTS.AxisRefMover[57].PlcToNc <-> Inputs/FromPlc
//   XtsTransport/XtsTransport Instance <-> NC-Task 1/Axes/Mover Axis 58
//     PLC_1 Inputs/GVL_XTS.AxisRefMover[58].NcToPlc <-> Outputs/ToPlc
//     PLC_1 Outputs/GVL_XTS.AxisRefMover[58].PlcToNc <-> Inputs/FromPlc
//   XtsTransport/XtsTransport Instance <-> NC-Task 1/Axes/Mover Axis 59
//     PLC_1 Inputs/GVL_XTS.AxisRefMover[59].NcToPlc <-> Outputs/ToPlc
//     PLC_1 Outputs/GVL_XTS.AxisRefMover[59].PlcToNc <-> Inputs/FromPlc
//   XtsTransport/XtsTransport Instance <-> NC-Task 1/Axes/Mover Axis 6
//     PLC_1 Inputs/GVL_XTS.AxisRefMover[6].NcToPlc <-> Outputs/ToPlc
//     PLC_1 Outputs/GVL_XTS.AxisRefMover[6].PlcToNc <-> Inputs/FromPlc
//   XtsTransport/XtsTransport Instance <-> NC-Task 1/Axes/Mover Axis 60
//     PLC_1 Inputs/GVL_XTS.AxisRefMover[60].NcToPlc <-> Outputs/ToPlc
//     PLC_1 Outputs/GVL_XTS.AxisRefMover[60].PlcToNc <-> Inputs/FromPlc
//   XtsTransport/XtsTransport Instance <-> NC-Task 1/Axes/Mover Axis 61
//     PLC_1 Inputs/GVL_XTS.AxisRefMover[61].NcToPlc <-> Outputs/ToPlc
//     PLC_1 Outputs/GVL_XTS.AxisRefMover[61].PlcToNc <-> Inputs/FromPlc
//   XtsTransport/XtsTransport Instance <-> NC-Task 1/Axes/Mover Axis 62
//     PLC_1 Inputs/GVL_XTS.AxisRefMover[62].NcToPlc <-> Outputs/ToPlc
//     PLC_1 Outputs/GVL_XTS.AxisRefMover[62].PlcToNc <-> Inputs/FromPlc
//   XtsTransport/XtsTransport Instance <-> NC-Task 1/Axes/Mover Axis 63
//     PLC_1 Inputs/GVL_XTS.AxisRefMover[63].NcToPlc <-> Outputs/ToPlc
//     PLC_1 Outputs/GVL_XTS.AxisRefMover[63].PlcToNc <-> Inputs/FromPlc
//   XtsTransport/XtsTransport Instance <-> NC-Task 1/Axes/Mover Axis 64
//     PLC_1 Inputs/GVL_XTS.AxisRefMover[64].NcToPlc <-> Outputs/ToPlc
//     PLC_1 Outputs/GVL_XTS.AxisRefMover[64].PlcToNc <-> Inputs/FromPlc
//   XtsTransport/XtsTransport Instance <-> NC-Task 1/Axes/Mover Axis 65
//     PLC_1 Inputs/GVL_XTS.AxisRefMover[65].NcToPlc <-> Outputs/ToPlc
//     PLC_1 Outputs/GVL_XTS.AxisRefMover[65].PlcToNc <-> Inputs/FromPlc
//   XtsTransport/XtsTransport Instance <-> NC-Task 1/Axes/Mover Axis 66
//     PLC_1 Inputs/GVL_XTS.AxisRefMover[66].NcToPlc <-> Outputs/ToPlc
//     PLC_1 Outputs/GVL_XTS.AxisRefMover[66].PlcToNc <-> Inputs/FromPlc
//   XtsTransport/XtsTransport Instance <-> NC-Task 1/Axes/Mover Axis 67
//     PLC_1 Inputs/GVL_XTS.AxisRefMover[67].NcToPlc <-> Outputs/ToPlc
//     PLC_1 Outputs/GVL_XTS.AxisRefMover[67].PlcToNc <-> Inputs/FromPlc
//   XtsTransport/XtsTransport Instance <-> NC-Task 1/Axes/Mover Axis 68
//     PLC_1 Inputs/GVL_XTS.AxisRefMover[68].NcToPlc <-> Outputs/ToPlc
//     PLC_1 Outputs/GVL_XTS.AxisRefMover[68].PlcToNc <-> Inputs/FromPlc
//   XtsTransport/XtsTransport Instance <-> NC-Task 1/Axes/Mover Axis 69
//     PLC_1 Inputs/GVL_XTS.AxisRefMover[69].NcToPlc <-> Outputs/ToPlc
//     PLC_1 Outputs/GVL_XTS.AxisRefMover[69].PlcToNc <-> Inputs/FromPlc
//   XtsTransport/XtsTransport Instance <-> NC-Task 1/Axes/Mover Axis 7
//     PLC_1 Inputs/GVL_XTS.AxisRefMover[7].NcToPlc <-> Outputs/ToPlc
//     PLC_1 Outputs/GVL_XTS.AxisRefMover[7].PlcToNc <-> Inputs/FromPlc
//   XtsTransport/XtsTransport Instance <-> NC-Task 1/Axes/Mover Axis 70
//     PLC_1 Inputs/GVL_XTS.AxisRefMover[70].NcToPlc <-> Outputs/ToPlc
//     PLC_1 Outputs/GVL_XTS.AxisRefMover[70].PlcToNc <-> Inputs/FromPlc
//   XtsTransport/XtsTransport Instance <-> NC-Task 1/Axes/Mover Axis 71
//     PLC_1 Inputs/GVL_XTS.AxisRefMover[71].NcToPlc <-> Outputs/ToPlc
//     PLC_1 Outputs/GVL_XTS.AxisRefMover[71].PlcToNc <-> Inputs/FromPlc
//   XtsTransport/XtsTransport Instance <-> NC-Task 1/Axes/Mover Axis 72
//     PLC_1 Inputs/GVL_XTS.AxisRefMover[72].NcToPlc <-> Outputs/ToPlc
//     PLC_1 Outputs/GVL_XTS.AxisRefMover[72].PlcToNc <-> Inputs/FromPlc
//   XtsTransport/XtsTransport Instance <-> NC-Task 1/Axes/Mover Axis 73
//     PLC_1 Inputs/GVL_XTS.AxisRefMover[73].NcToPlc <-> Outputs/ToPlc
//     PLC_1 Outputs/GVL_XTS.AxisRefMover[73].PlcToNc <-> Inputs/FromPlc
//   XtsTransport/XtsTransport Instance <-> NC-Task 1/Axes/Mover Axis 74
//     PLC_1 Inputs/GVL_XTS.AxisRefMover[74].NcToPlc <-> Outputs/ToPlc
//     PLC_1 Outputs/GVL_XTS.AxisRefMover[74].PlcToNc <-> Inputs/FromPlc
//   XtsTransport/XtsTransport Instance <-> NC-Task 1/Axes/Mover Axis 75
//     PLC_1 Inputs/GVL_XTS.AxisRefMover[75].NcToPlc <-> Outputs/ToPlc
//     PLC_1 Outputs/GVL_XTS.AxisRefMover[75].PlcToNc <-> Inputs/FromPlc
//   XtsTransport/XtsTransport Instance <-> NC-Task 1/Axes/Mover Axis 76
//     PLC_1 Inputs/GVL_XTS.AxisRefMover[76].NcToPlc <-> Outputs/ToPlc
//     PLC_1 Outputs/GVL_XTS.AxisRefMover[76].PlcToNc <-> Inputs/FromPlc
//   XtsTransport/XtsTransport Instance <-> NC-Task 1/Axes/Mover Axis 77
//     PLC_1 Inputs/GVL_XTS.AxisRefMover[77].NcToPlc <-> Outputs/ToPlc
//     PLC_1 Outputs/GVL_XTS.AxisRefMover[77].PlcToNc <-> Inputs/FromPlc
//   XtsTransport/XtsTransport Instance <-> NC-Task 1/Axes/Mover Axis 78
//     PLC_1 Inputs/GVL_XTS.AxisRefMover[78].NcToPlc <-> Outputs/ToPlc
//     PLC_1 Outputs/GVL_XTS.AxisRefMover[78].PlcToNc <-> Inputs/FromPlc
//   XtsTransport/XtsTransport Instance <-> NC-Task 1/Axes/Mover Axis 79
//     PLC_1 Inputs/GVL_XTS.AxisRefMover[79].NcToPlc <-> Outputs/ToPlc
//     PLC_1 Outputs/GVL_XTS.AxisRefMover[79].PlcToNc <-> Inputs/FromPlc
//   XtsTransport/XtsTransport Instance <-> NC-Task 1/Axes/Mover Axis 8
//     PLC_1 Inputs/GVL_XTS.AxisRefMover[8].NcToPlc <-> Outputs/ToPlc
//     PLC_1 Outputs/GVL_XTS.AxisRefMover[8].PlcToNc <-> Inputs/FromPlc
//   XtsTransport/XtsTransport Instance <-> NC-Task 1/Axes/Mover Axis 80
//     PLC_1 Inputs/GVL_XTS.AxisRefMover[80].NcToPlc <-> Outputs/ToPlc
//     PLC_1 Outputs/GVL_XTS.AxisRefMover[80].PlcToNc <-> Inputs/FromPlc
//   XtsTransport/XtsTransport Instance <-> NC-Task 1/Axes/Mover Axis 81
//     PLC_1 Inputs/GVL_XTS.AxisRefMover[81].NcToPlc <-> Outputs/ToPlc
//     PLC_1 Outputs/GVL_XTS.AxisRefMover[81].PlcToNc <-> Inputs/FromPlc
//   XtsTransport/XtsTransport Instance <-> NC-Task 1/Axes/Mover Axis 82
//     PLC_1 Inputs/GVL_XTS.AxisRefMover[82].NcToPlc <-> Outputs/ToPlc
//     PLC_1 Outputs/GVL_XTS.AxisRefMover[82].PlcToNc <-> Inputs/FromPlc
//   XtsTransport/XtsTransport Instance <-> NC-Task 1/Axes/Mover Axis 83
//     PLC_1 Inputs/GVL_XTS.AxisRefMover[83].NcToPlc <-> Outputs/ToPlc
//     PLC_1 Outputs/GVL_XTS.AxisRefMover[83].PlcToNc <-> Inputs/FromPlc
//   XtsTransport/XtsTransport Instance <-> NC-Task 1/Axes/Mover Axis 84
//     PLC_1 Inputs/GVL_XTS.AxisRefMover[84].NcToPlc <-> Outputs/ToPlc
//     PLC_1 Outputs/GVL_XTS.AxisRefMover[84].PlcToNc <-> Inputs/FromPlc
//   XtsTransport/XtsTransport Instance <-> NC-Task 1/Axes/Mover Axis 85
//     PLC_1 Inputs/GVL_XTS.AxisRefMover[85].NcToPlc <-> Outputs/ToPlc
//     PLC_1 Outputs/GVL_XTS.AxisRefMover[85].PlcToNc <-> Inputs/FromPlc
//   XtsTransport/XtsTransport Instance <-> NC-Task 1/Axes/Mover Axis 86
//     PLC_1 Inputs/GVL_XTS.AxisRefMover[86].NcToPlc <-> Outputs/ToPlc
//     PLC_1 Outputs/GVL_XTS.AxisRefMover[86].PlcToNc <-> Inputs/FromPlc
//   XtsTransport/XtsTransport Instance <-> NC-Task 1/Axes/Mover Axis 87
//     PLC_1 Inputs/GVL_XTS.AxisRefMover[87].NcToPlc <-> Outputs/ToPlc
//     PLC_1 Outputs/GVL_XTS.AxisRefMover[87].PlcToNc <-> Inputs/FromPlc
//   XtsTransport/XtsTransport Instance <-> NC-Task 1/Axes/Mover Axis 88
//     PLC_1 Inputs/GVL_XTS.AxisRefMover[88].NcToPlc <-> Outputs/ToPlc
//     PLC_1 Outputs/GVL_XTS.AxisRefMover[88].PlcToNc <-> Inputs/FromPlc
//   XtsTransport/XtsTransport Instance <-> NC-Task 1/Axes/Mover Axis 89
//     PLC_1 Inputs/GVL_XTS.AxisRefMover[89].NcToPlc <-> Outputs/ToPlc
//     PLC_1 Outputs/GVL_XTS.AxisRefMover[89].PlcToNc <-> Inputs/FromPlc
//   XtsTransport/XtsTransport Instance <-> NC-Task 1/Axes/Mover Axis 9
//     PLC_1 Inputs/GVL_XTS.AxisRefMover[9].NcToPlc <-> Outputs/ToPlc
//     PLC_1 Outputs/GVL_XTS.AxisRefMover[9].PlcToNc <-> Inputs/FromPlc
//   XtsTransport/XtsTransport Instance <-> NC-Task 1/Axes/Mover Axis 90
//     PLC_1 Inputs/GVL_XTS.AxisRefMover[90].NcToPlc <-> Outputs/ToPlc
//     PLC_1 Outputs/GVL_XTS.AxisRefMover[90].PlcToNc <-> Inputs/FromPlc
//   XtsTransport/XtsTransport Instance <-> NC-Task 1/Axes/Mover Axis 91
//     PLC_1 Inputs/GVL_XTS.AxisRefMover[91].NcToPlc <-> Outputs/ToPlc
//     PLC_1 Outputs/GVL_XTS.AxisRefMover[91].PlcToNc <-> Inputs/FromPlc
//   XtsTransport/XtsTransport Instance <-> NC-Task 1/Axes/Mover Axis 92
//     PLC_1 Inputs/GVL_XTS.AxisRefMover[92].NcToPlc <-> Outputs/ToPlc
//     PLC_1 Outputs/GVL_XTS.AxisRefMover[92].PlcToNc <-> Inputs/FromPlc
//   XtsTransport/XtsTransport Instance <-> NC-Task 1/Axes/Mover Axis 93
//     PLC_1 Inputs/GVL_XTS.AxisRefMover[93].NcToPlc <-> Outputs/ToPlc
//     PLC_1 Outputs/GVL_XTS.AxisRefMover[93].PlcToNc <-> Inputs/FromPlc
//   XtsTransport/XtsTransport Instance <-> NC-Task 1/Axes/Mover Axis 94
//     PLC_1 Inputs/GVL_XTS.AxisRefMover[94].NcToPlc <-> Outputs/ToPlc
//     PLC_1 Outputs/GVL_XTS.AxisRefMover[94].PlcToNc <-> Inputs/FromPlc
//   XtsTransport/XtsTransport Instance <-> NC-Task 1/Axes/Mover Axis 95
//     PLC_1 Inputs/GVL_XTS.AxisRefMover[95].NcToPlc <-> Outputs/ToPlc
//     PLC_1 Outputs/GVL_XTS.AxisRefMover[95].PlcToNc <-> Inputs/FromPlc
//   XtsTransport/XtsTransport Instance <-> NC-Task 1/Axes/Mover Axis 96
//     PLC_1 Inputs/GVL_XTS.AxisRefMover[96].NcToPlc <-> Outputs/ToPlc
//     PLC_1 Outputs/GVL_XTS.AxisRefMover[96].PlcToNc <-> Inputs/FromPlc
//   XtsTransport/XtsTransport Instance <-> NC-Task 1/Axes/Mover Axis 97
//     PLC_1 Inputs/GVL_XTS.AxisRefMover[97].NcToPlc <-> Outputs/ToPlc
//     PLC_1 Outputs/GVL_XTS.AxisRefMover[97].PlcToNc <-> Inputs/FromPlc
//   XtsTransport/XtsTransport Instance <-> NC-Task 1/Axes/Mover Axis 98
//     PLC_1 Inputs/GVL_XTS.AxisRefMover[98].NcToPlc <-> Outputs/ToPlc
//     PLC_1 Outputs/GVL_XTS.AxisRefMover[98].PlcToNc <-> Inputs/FromPlc
//   XtsTransport/XtsTransport Instance <-> NC-Task 1/Axes/Mover Axis 99
//     PLC_1 Inputs/GVL_XTS.AxisRefMover[99].NcToPlc <-> Outputs/ToPlc
//     PLC_1 Outputs/GVL_XTS.AxisRefMover[99].PlcToNc <-> Inputs/FromPlc
//   XtsTransport/XtsTransport Instance <-> NC-Task 1/Objects/Group1 (CA Group)
//     PLC_1 Inputs/GVL_XTS.CaGroupRef.NcToPlc/CA <-> Group Outputs/ToPLC
//     PLC_1 Outputs/GVL_XTS.CaGroupRef.PlcToNc/CA <-> Group Inputs/FromPLC

CONFIGURATION XtsTransport
    RESOURCE PLC ON TwinCAT3
        TASK PLC_1(INTERVAL := T#1ms, PRIORITY := 15);
        PROGRAM MAPPING_in WITH PLC_1 : MAPPING_in;
        PROGRAM MAIN_APP WITH PLC_1 : MAIN_APP;
        PROGRAM MAIN WITH PLC_1 : MAIN;
        PROGRAM MAPPING_out WITH PLC_1 : MAPPING_out;
    END_RESOURCE
END_CONFIGURATION

// ---- APPLICATION/_types/Application/E_APP_CHECK.TcDUT
{attribute 'qualified_only'}
{attribute 'strict'}
{attribute 'to_string'}
TYPE E_APP_CHECK :
(
  CHECK_INIT,

  INVALID_CTRL_POINTER,
  INVALID_STATE_POINTER,
  INVALID_INSTANCE_CONTROL_REFERENCE,
  INVALID_INSTANCE_STATE_REFERENCE,
	INVALID_TRANSPORT_CTRL_POINTER    := 10,
	INVALID_TRANSPORT_STATE_POINTER   := 20,
	INVALID_COLLECTOR_INTERFACE       := 30,
  INVALID_PROCESS_LIST_INTERFACE    := 40,

  CHECK_DONE := 10000

)UINT;
END_TYPE

// ---- APPLICATION/_types/Application/E_APP_VARIANT.TcDUT
{attribute 'qualified_only'}
{attribute 'strict'}
{attribute 'to_string'}
TYPE E_APP_VARIANT :
(
  VARIANT_INVALID,
	VARIANT_OUTPUT_24,
  VARIANT_OUTPUT_CLAMP
);
END_TYPE

// ---- APPLICATION/_types/Application/ST_APP_CTRL.TcDUT
TYPE ST_APP_CTRL :
STRUCT
  Cmd       : E_INSTANCE_CMD;
  Variant   : E_APP_VARIANT;
END_STRUCT
END_TYPE

// ---- APPLICATION/_types/Application/ST_APP_STATE.TcDUT
TYPE ST_APP_STATE :
STRUCT
  AppInit             : E_PROGRESS;
  AppState            : E_INSTANCE_STATE;
END_STRUCT
END_TYPE

// ---- APPLICATION/_types/Collector/E_PROCESS_CTRL.TcDUT
{attribute 'qualified_only'}
{attribute 'strict'}
{attribute 'to_string'}
TYPE E_PROCESS_CTRL :
(
  PROCESS_INIT              := 10,
  PROCESS_DISABLE           := 20,
  PROCESS_ENABLE            := 30,
  PROCESS_STATIONS_INFEED,

  PROCESS_STATIONS_ENTER    := 40,
  PROCESS_STATIONS_SEND,

  PROCESS_START             := 60,
  PROCESS_DONE              := 70,
  PROCESS_STATIONS_OUTFEED  := 80
);
END_TYPE

// ---- APPLICATION/_types/Instance/E_INSTANCE.TcDUT
{attribute 'qualified_only'}
//{attribute 'strict'}
{attribute 'to_string'}
TYPE E_INSTANCE :
(
  // process identifiers as enum, 
  // this enum must not have gaps!
  INVALID,
  PROCESS_CONDUCTOR,
  BUFFER_INFEED,                    // process for getting the job from transfersystem
  INFEED,                           // process for getting workpieces from transfersystem
  BUFFER_OUTFEED,                   // process for dealing movers into robot outfeed with no gaps
  OUTFEED_ROBOT_R1,                 // process for robot outfeed (12 movers)
  OUTFEED_ROBOT_R2,                 // process for robot outfeed (12 movers)
  //SENDER_SLOW,                    // process for slowing down movers
  SENDER_FAST,                      // process for accelerating movers to return with max velo
  SENDER_BUFFER_INFEED,             // process for dealing movers into BUFFER_INFEED, since the curve is vertical, there has to be room when movers are set in motion
  INSTANCE_MAX
)UINT;
END_TYPE

// ---- APPLICATION/_types/Instance/E_INSTANCE_CHECK.TcDUT
{attribute 'qualified_only'}
{attribute 'strict'}
{attribute 'to_string'}
TYPE E_INSTANCE_CHECK :
(
  CHECK_INIT,

	INVALID_INTERFACE_POINTER := 10,
  INVALID_INSTANCE_CONTROL_REFERENCE,
  INVALID_INSTANCE_STATE_REFERENCE,
  INVALID_PROCESS_ID_ZERO,
  INVALID_PROCESS_ID_MAX,
  INVALID_PROCESS_ID_NOTEQUAL_COLLECTOR_ID,
  INVALID_INDEX_IN_LIST,

  CHECK_DONE := 10000
)UINT;
END_TYPE

// ---- APPLICATION/_types/Instance/E_INSTANCE_STATE.TcDUT
{attribute 'qualified_only'}
//{attribute 'strict'}
{attribute 'to_string'}
TYPE E_INSTANCE_STATE :
(
  NULL,
	INVALID,
  INIT,
  DISABLED,
  DETECTION,
  ENABLED,
  WORKING,
  PROCEEDING,
  FINISH,
  CLEARED
)UINT;
END_TYPE

// ---- MSG/types/ST_Message.TcDUT
TYPE ST_Message :
STRUCT
  eType         : e_MessageType;
  eDevice       : e_Device;
  eSubdevice    : e_SubDevice;
  {attribute 'displaymode':='hex'}
  iErrorNumber  : LINT;
  tTime         : STRING(24);
  sText         : STRING(127);
END_STRUCT
END_TYPE

// ---- XTS/CaGroup/types/E_CA_GROUP_STATE.TcDUT
// {attribute 'qualified_only'}
// {attribute 'strict'}
{attribute 'to_string'}
TYPE E_CA_GROUP_STATE :
(
  // replicated from MC_GROUP_STATE for getting to_string() functionality
	mcGroupStateInvalid   :=0, 
  mcGroupStateDisabled  :=1, 
  mcGroupStateStandby   :=2, 
  mcGroupStateMoving    :=3, 
  mcGroupStateStopping  :=4, 
  mcGroupStateErrorStop :=5, 
  mcGroupStateHoming    :=6, 
  mcGroupStateNotReady  :=7, 
  mcGroupStateSuspended :=8 
)UINT;
END_TYPE

// ---- XTS/CaGroup/types/E_GROUP_CHECK.TcDUT
{attribute 'qualified_only'}
{attribute 'to_string'}
TYPE E_GROUP_CHECK :
(
  CHECK_NULL,
  CHECK_GROUP_REF_INVALID := 10,
  CHECK_AXIS_REF_INVALID,
  CHECK_CTRL_INVALID,
  CHECK_STATE_INVALID,
  CHECK_Mover_ITF_REF_INVALID,
  CHECK_XPU_INFO_REF_INVALID,


  CHECK_ERROR             :=  9000,
  CHECK_DONE              := 10000
)UINT;
END_TYPE

// ---- XTS/Mover/types/E_MOVER_CTRL.TcDUT
{attribute 'qualified_only'}
{attribute 'strict'}
{attribute 'to_string'}
TYPE E_MOVER_CTRL :
(
  MOVER_NULL,               // initial value at startup, used for change of order or retrigger
  MOVER_ENABLE,             // sets MC_Power.Enable
  MOVER_DISABLE,            // removes MC_Power.Enable
  MOVER_MOVE_TO_POS,        // modulo absolute positioning with MC_MoveAbsolute, InTargetPosition check
  MOVER_MOVE_TO_POS_CA,     // modulo absolute positioning with MC_MoveAbsoluteCA, InTargetPosition check
  MOVER_SEND_TO_POS_CA,     // modulo absolute positioning with MC_MoveAbsoluteCA, done after moving ReleaseDistance
  MOVER_HALT,               // halts mover; by use of MC_Halt mover is set passive in CA group
  MOVER_GEAR_IN,            // GearIn for mover in standstill

  MOVER_GEAR_IN_POS_CA,     // GearInPosCA of mover; when FB_GearInPosCa is InSync --> order is done; check SyncDistance yourself and release mover with e_mover_order.mover_SendToPos
  MOVER_GEAR_OUT,           // gear out for mover
  MOVER_RESET               // MC_RESET for mover
)UINT;
END_TYPE

// ---- XTS/Mover/types/E_MOVER_STATE.TcDUT
{attribute 'qualified_only'}
{attribute 'to_string'}
TYPE E_MOVER_STATE :
(
  MOVER_NULL,               // initial value at startup, used for change of order or retrigger
  MOVER_ENABLE,             // sets MC_Power.Enable
  MOVER_DISABLE,            // removes MC_Power.Enable
  MOVER_MOVE_TO_POS,        // modulo absolute positioning with MC_MoveAbsolute, InTargetPosition check
  MOVER_MOVE_TO_POS_CA,     // modulo absolute positioning with MC_MoveAbsoluteCA, InTargetPosition check
  MOVER_SEND_TO_POS_CA,     // modulo absolute positioning with MC_MoveAbsoluteCA, done after moving ReleaseDistance
  MOVER_HALT,               // halts mover; by use of MC_Halt mover is set passive in CA group
  MOVER_GEAR_IN,            // GearIn for mover in standstill

  MOVER_GEAR_IN_POS_CA,     // GearInPosCA of mover; when FB_GearInPosCa is InSync --> order is done; check SyncDistance yourself and release mover with e_mover_order.mover_SendToPos
  MOVER_GEAR_OUT,           // gear out for mover
  MOVER_RESET               // MC_RESET for mover
)UINT;
END_TYPE

// ---- XTS/Mover/types/ST_MOVER_CTRL.TcDUT
{attribute 'pack_mode' := '2'}
TYPE ST_MOVER_CTRL :
STRUCT
  Cmd             : E_MOVER_CTRL;  // order to execute on mover
END_STRUCT
END_TYPE

// ---- XTS/Mover/types/ST_MOVER_INFO.TcDUT
{attribute 'pack_mode' := '2'}
TYPE ST_MOVER_INFO :
STRUCT
  bMoverEnabled           : BIT;    // Axis[i].Status.ControlLoopClosed
  bMoverError             : BIT;    // Axis[i].Status.Error
  bMoverCoupled           : BIT;    // Axis[i].Status.Coupled OR _fbGearInPosCa[i].InSync
  bMoverStandstill        : BIT;    // Axis[i].Status.NotMoving
  bMoverAvoidingCollision : BIT;    // Axis[i].NcToPlc.StateDWord2.0
  bMoverInTarget          : BIT;    // Axis[i].NcToPlc.ActPos == rLastSetPos[i]

  rModuloActPos           : REAL;   // TO_REAL(Axis[i].NcToPlc.ModuloActPos)
  rAbsActPos              : REAL;   // TO_REAL(Axis[i].NcToPlc.ActPos)
  rAbsTargetPos           : REAL;   // TO_REAL(rLastSetPos[i])
  rModuloTargetPos        : REAL;   // TO_REAL(Tc2_Math.LMOD(_rLastSetPos[i], _RailLength))

  nErrorId                : UDINT;
END_STRUCT
END_TYPE

// ---- XTS/Mover/types/ST_MOVER_STATE.TcDUT
{attribute 'pack_mode' := '2'}
TYPE ST_MOVER_STATE :
STRUCT
  State           : E_MOVER_STATE;  // ST_MOVER_CTRL.Cmd with added E_PROGRESS
  MasterId        : USINT;            // mirror NC AxisId of Master axis
END_STRUCT
END_TYPE

// ---- XTS/Mover/types/ST_MOVE_DATA.TcDUT
{attribute 'pack_mode' := '2'}
TYPE ST_MOVE_DATA :
STRUCT
  // HAUD 2024 03 14
  // some init data added for example
  rPos            : LREAL :=   2275.0;
  rVelo           : LREAL :=    500.0;
  rAcc            : LREAL :=   5000.0;
  rJerk           : LREAL := 500000.0;
  rGap            : LREAL :=    100.0;
  rOverride       : LREAL :=    100.0;
  rDelta          : LREAL :=      0.05;
  rDistance       : LREAL :=     25.0;
END_STRUCT
END_TYPE

// ---- XTS/Xpu/types/E_XPU_CTRL.TcDUT
{attribute 'strict'}
TYPE E_XPU_CTRL :
(
  XTS_CMD_NULL,
  XTS_CMD_INIT                  := 10,
  //XTS_CMD_READ_STN_CONFIG       := 20,
  XTS_IDLE                      := 30
)UINT;
END_TYPE

// ---- XTS/Xpu/types/E_XPU_INIT.TcDUT
{attribute 'to_string'}
TYPE E_XPU_INIT :
(
	INIT_START,
  INIT_ENVIRONMENT_OID            := 10,
  INIT_INFO_SERVER_ITF,
  INIT_INFO_SERVER_STATION_COUNT,
  INIT_INFO_SERVER_STATION_OID,
  INIT_CA_GROUP_OID               := 20,
  INIT_CA_GROUP_GET_OID,
  INIT_CA_GROUP_CHECK_OID,
  INIT_CA_GROUP_COM,
  INIT_PARAMETERSET_COUNT,
  INIT_PARAMETERSET_OID,
  INIT_PARAMETERSET_COM,
  INIT_PARAMETERSET_COM_NEXT,
  INIT_PROCESSING_UNIT_COM        := 30,
  INIT_PROCESSING_UNIT_PART_COUNT,
  INIT_PROCESSING_UNIT_PART_OID,
  INIT_PROCESSING_UNIT_TRACK_COUNT,
  INIT_PROCESSING_UNIT_TRACK_OID,
  INIT_PROCESSING_UNIT_MOVER_COUNT,
  INIT_PROCESSING_UNIT_MOVER_OID,
  INIT_PROCESSING_UNIT_TASK_COUNT,
  INIT_PROCESSING_UNIT_TASK_OID,
  INIT_TRACK_COM                  := 50,
  INIT_PART_COM                   := 60,
  INIT_PART_MODULE_COUNT,
  INIT_PART_MODULE_OID,
  INIT_PART_MODULE_COM,
  INIT_PART_MODULE_COM_NEXT,
  INIT_MOVER_COM                  := 70,
  INIT_MOVER_COM_NEXT,
  INIT_NCT_CONTROLLER_OID         := 80,
  INIT_NCT_CONTROLLER_COM,
  INIT_NCT_BASE_UNIT_COUNT,
  INIT_NCT_BASE_UNIT_ITF,
  INIT_NCT_BASE_UNIT_NEXT,
  INIT_DATA_GET                   := 90,
  INIT_DATA_CHECK,
  INIT_DONE                       := 100
)UINT;
END_TYPE

// ---- XTS/Xpu/types/E_XPU_STATE.TcDUT
{attribute 'to_string'}
TYPE E_XPU_STATE :
(
  XTS_NULL,
  XTS_INVALID,
  XTS_INIT                      := 10,    // initialize XPU
  XTS_STATION_INFO_READ         := 20,    // get Station information from Xpu
  XTS_IDLE                      := 30
)UINT;
END_TYPE

// ---- XTS/Xpu/types/ST_XPU_CTRL.TcDUT
{attribute 'pack_mode' := '2'}
TYPE ST_XPU_CTRL :
STRUCT
  Cmd             : E_XPU_CTRL;
END_STRUCT
END_TYPE

// ---- XTS/Xpu/types/ST_XPU_INFO.TcDUT
{attribute 'pack_mode' := '2'}
TYPE ST_XPU_INFO :
STRUCT
  AllPositionsValid   : BIT;
  IdDetectionError    : BIT;
  IdDetectionValid    : BIT;
  IdDetectionActive   : BIT;

  OperationMode       : UINT;

  IdDetectionMode           : UINT;
  MoverPositionAssignement  : UINT;

  nDetectedAxisCount  : UINT;
  nExpectedAxisCount  : UINT;

  nParameterSetCount  : UINT;
  
END_STRUCT
END_TYPE

// ---- XTS/XtsStation/_types/E_STATION_STATE.TcDUT
{attribute 'qualified_only'}
{attribute 'to_string'}
TYPE E_STATION_STATE :
(
	STATION_NO_INIT,                // startup state after power on, first cycle Init of station, switches to INIT when done

  STATION_INIT,                   // CONTINUE to DISABLE
                                  // State.MoverId deleted

  STATION_DISABLE         := 10,  // + CTRL.STATION_ENABLE  --> CONTINUE to DETECT_MOVER 
                                  // station is empty, no mover is handled, check enable from ctrl

  STATION_ENABLE,                 // init of work vars, check enable from ctrl

  STATION_DETECT_MOVER,           // (QueueCount > 0)       --> CONTINUE to MOVER_ENTER

  STATION_MOVER_ENTER     := 20,  // + CTRL.MOVER_ENTER     --> CONTINUE to PROCESS_START
                                  // + CTRL.MOVER_SEND      --> CONTINUE to MOVER_OUT
                                  // mover asking for entry

  STATION_MOVER_IN_TARGET,        // (MoveToPos==TRUE)      --> CONTINUE to PROCESS_START
                                  // mover is moving to PosWait + PosStop[_nNest]

  STATION_PROCESS_START   := 30,  // + CTRL.PROCESS_START   --> CONTINUE to PROCESS_START
                                  // + CTRL.PROCESS_DONE    --> CONTINUE to CHECK
                                  // wait until process started

  STATION_PROCESS_DONE,           // + CTRL.PROCESS_DONE    --> CONTINUE to CHECK
                                  // wait until process done

  STATION_CHECK           := 40,  // check for next nest in mask, 
                                  // (mask<>0) --> CHECK_NEST
                                  // (mask==0) --> MOVER_OUT

  STATION_CHECK_NEST,             // + CTRL.MOVER_ENTER     --> CONTINUE to MOVER_IN_TARGET
                                  // get next nest position

  STATION_MOVER_OUT       := 50,  // + CTRL.MOVER_OUT       --> CONTINUE to MOVER_RELEASE
                                  // mover asking to leave

  STATION_MOVER_RELEASE,          // (MoverSendToPos==TRUE) --> CONTINUE to MOVER_GONE
                                  // mover is released + check if release distance is passed

  STATION_MOVER_WRITE_TARGET,     // worker state to write mover ticket

  STATION_MOVER_GONE      := 60,  // + CTRL.MOVER_GONE      --> CONTINUE to INIT
                                  // mover out of station, enter mover in target station list


  STATION_ERROR_NULL      := 127,
  STATION_ERROR_LIST_GET_HEAD_FAULT,    // fatal error in linked list, must never occurr, must be debugged
  STATION_ERROR_LIST_REMOVE_HEAD_FAULT, // fatal error in linked list, must never occurr, must be debugged
  STATION_ERROR_LIST_ADD_TAIL_FAULT,    // fatal error in linked list, must never occurr, must be debugged

  STATION_ERROR_LIST_STATION_ID_WRONG,  // ticket data in Queue contains wrong Station Id, can be overruled by ctrl

  STATION_ERROR_LIST_MOVER_ID_INVALID,  // fatal error in ticket data, MoverId is out of range, must be fixed by ctrl, must be debugged

  STATION_ERROR_INFEED_ERROR,           // motion error during movement, retry must be triggered by ctrl
  STATION_ERROR_OUTFEED_ERROR,          // motion error during movement, retry by ctrl OR leave by ctrl

  STATION_ERROR_OUTFEED_TARGET_INVALID, // ticket data for nTargetStation is not plausible, can be fixed by ctrl

  STATION_ERROR_FATAL     := 255 // the thing that must not be, all fatal errors end up here
)USINT;
END_TYPE

// ---- XTS/XtsStation/_types/ST_STATION_LIST_RESULT.TcDUT
TYPE ST_STATION_LIST_RESULT :
STRUCT
  wState    : WORD;   // wState == 0 --> all ok
  nIndex    : ULINT;
  stData    : ST_STATION_MOVER_DATA;  // copy of list entry
END_STRUCT
END_TYPE

// ---- XTS/XtsStation/_types/ST_STATION_MOVER_DATA.TcDUT
{attribute 'pack_mode' := '2'}
TYPE ST_STATION_MOVER_DATA :
STRUCT
  nMoverId        : USINT;  // who am I?  !! MUST be correct !! - movement to base position sets everything in order, DO NOT manipulate!
  nTargetStation  : USINT;  // where shall I be? used for double checking with StationId at infeed of mover into station

  {attribute 'displaymode':='bin'}
  nMask           : BYTE;   // how many of you are there? (1 = default, no action required)

  rOffset         : REAL;   // offset for use in work flow !! added to static mover offset for every nest(bit) in nMask!!
END_STRUCT
END_TYPE

// ---- XTS/XtsStation/_types/ST_STATION_STATE.TcDUT
{attribute 'pack_mode' := '2'}
TYPE ST_STATION_STATE :
STRUCT
  eState          : E_STATION_STATE;
  {attribute 'displaymode':='bin'}
  nMask           : BYTE;
  nMoverId        : USINT;
  rMoverModPos    : LREAL;            // modulo position of detected mover
  nQueue          : USINT;            // queue count for station
END_STRUCT
END_TYPE

// ---- XTS/_Visualization/types/ST_XPU_STRINGS.TcDUT
TYPE ST_XPU_STRINGS :
STRUCT
  sXpuState       ,
  sXpuResult      ,
  sXpuCyclicCheck ,
  sXpuOpMode      ,
  sXpuMoverId_DetectionMode,
  sXpuMoverPosAssignement : STRING(30) := 'NULL';
END_STRUCT
END_TYPE

// ---- APPLICATION/GVL_APPLICATION.TcGVL
VAR_GLOBAL CONSTANT
  MAX_PROCESS         : E_INSTANCE := E_INSTANCE.SENDER_BUFFER_INFEED;
END_VAR
{attribute 'qualified_only'}
VAR_GLOBAL
  //-----------------------------------------------------------------------------------------------
  // fb_Application
  //
  //  is the part you'll find in ExternControl PLC
  //-----------------------------------------------------------------------------------------------
  //-----------------------------------------------------------------------------------------------
  //-----------------------------------------------------------------------------------------------
  AppControl            : ST_APP_CTRL;
  AppState              : ST_APP_STATE;

  //-----------------------------------------------------------------------------------------------
  // Process instances
  //  - processes are similar but also different, hence working with inheritance of fb_Instance
  //  - change/check here if you need a process procedure that matches your use case
  //-----------------------------------------------------------------------------------------------
  BufferInfeed          : fb_BufferInfeed;        // prepare movers to enter infeed station
  Infeed                : fb_Infeed;              // infeed into XTS, transfersystem drops its load here
  BufferOutfeed         : fb_BufferOutfeed;  // feeds 24 Mover into 2 processes (12 each), no gaps
  Outfeed_R1            : fb_Outfeed;        // unloads 12 mover
  Outfeed_R2            : fb_Outfeed;        // unloads 12 mover
  SenderFast            : fb_SenderBuffer;   // every passing mover is accelersted to max velo
  SenderBufferInfeed    : fb_SenderBuffer;   // checks if there is room for 12-x mover, sends mover to BufferInfeed for a new round


  //-----------------------------------------------------------------------------------------------
  // fb_Instance control and state
  //  - structs are used in fb_Application as reference 
  //-----------------------------------------------------------------------------------------------
  InstanceCtrl          : ARRAY[1..MAX_PROCESS] OF ST_INSTANCE_CTRL;
  InstanceState         : ARRAY[1..MAX_PROCESS] OF ST_INSTANCE_STATE;


  //-----------------------------------------------------------------------------------------------
  // Linked List instances
  //  - THIS example only uses the linked list in fb_BufferInfeed 
  //    as buffered input from an extern transfersystem
  //-----------------------------------------------------------------------------------------------
  ProcessList           : ARRAY[1..MAX_PROCESS] OF fb_Process_LinkedList; // information transfer between processes
  ItfProcessList        : ARRAY[1..MAX_PROCESS] OF I_Process_LinkedList;      // use this interface in your function blocks


  //-----------------------------------------------------------------------------------------------
  // Collector instances
  //
  //  - layer for grouping parallel XtsStations for process handshakes
  //-----------------------------------------------------------------------------------------------
  //  - fb_ProcessCollector:
  //    - uses .ProcessCtrl and .ProcessState for handshakes with application
  //
  //    - .ActivateStation is evaluated after enabling infeed in state 
  //      E_PROCESS_STATE.PROCESS_DISABLE:/E_PROGRESS.PROGRESS_BUSY:
  //      
  //    - ST_PROCESS_STATE:
  //      - contains 3 enumerations for you to check
  //      - State           : E_PROCESS_STATE;
  //        - main state for handshakes
  //
  //      - Result          : E_PROGRESS;
  //        - substate for checks during handshake; 
  //          PROGRESS_BUSY --> handshakes are accepted (see fb_ProcessCollecotr.Cycle())
  //
  //      - Check           : E_PROCESS_CHECK;
  //        - cyclic pointer check: use this on startup of your application
  //
  //    - inherits fb_StationCollector
  //-----------------------------------------------------------------------------------------------
  ProcessCollector      : ARRAY[1..MAX_PROCESS] OF fb_ProcessCollector;       // grouping of XtsStations
  ItfProcessCollector   : ARRAY[1..MAX_PROCESS] OF I_ProcessCollector;        // interface for use in your function blocks like BufferInfeed etc.


  //-----------------------------------------------------------------------------------------------
  // cyclic linked lists
  //
  //  - fb_LinkedListCtrl
  //    - is controlled via Ctrl/State pair
  //    - provides I_Process_LinkedList for use in conected class
  //-----------------------------------------------------------------------------------------------
  TicketControl         : fb_Process_LinkedListCtrl;
  TicketList            : fb_Process_LinkedList;
  TicketListControl     : ST_LIST_CTRL;
  TicketListState       : ST_LIST_STATE;
  TicketListDataInput   : ST_LIST_NODE_DATA;   // datafield for you to write(add) your data
  TicketListDataOutput  : ST_LIST_NODE_DATA;   // datafield for you to read (get) your data


  //-----------------------------------------------------------------------------------------------
  // Distribution of LinkedList ticket
  //
  //  - fb_ProcessConductor extends fb_Instance
  //    - is controlled via instance Ctrl/State pair
  //    - consumes I_Process_LinkedList for moving 
  //      the ticket from the cyclic list into the process list of ST_PROCESS_DATA.nProcessId
  //-----------------------------------------------------------------------------------------------
  ProcessConductor      : fb_ProcessConductor;
END_VAR

// ---- XTS/GVL_XTS.TcGVL
{attribute 'qualified_only'}
VAR_GLOBAL
  //---------------------------------------------------------------------------
  // XTS Station
  //  - handshakes mover in station with extern control
  //  - station parameters (positions, gap, dyn. constraints, description...)
  StationStart        : ST_STATION_PARAMETER;   // Xts transport is sending all mover to this position (CMD_TRANSPORT_START)
  StationStartIndex   : UINT := 52;              // index of XtsStation where all movers are entered into linked list.

  // station handshaking with mover and extern process
  // station sends mover to target station/WaitPos
  // station adds mover data to LinkedList.AddTail() of target station
  Station             : ARRAY[1..MAX_STATION] OF fb_StationProcess;
  StationGearIn       : ARRAY[1..MAX_STATION] OF fb_StationGearInPos;

  StationList         : ARRAY[1..MAX_STATION] OF fb_Station_LinkedList;

  StationQueue        : ARRAY[1..MAX_STATION]    OF 
                        ARRAY[1..MAX_LIST_NODES] OF ST_STATION_MOVER_DATA;

  // interface for access to List methods
  StationListItf      : ARRAY[1..MAX_STATION] OF I_Station_LinkedList;

  // interface for access to station methods
  StationCtrlItf      : ARRAY[1..MAX_STATION] OF I_XtsTransport_Station;

  // ctrl / state datafields for extern control
  StationCtrl         : ARRAY[1..MAX_STATION] OF ST_STATION_CTRL;   // control for extern to write, you can do whatever you want as long as you do as I say
  StationState        : ARRAY[1..MAX_STATION] OF ST_STATION_STATE;  // state for extern to read, this is what I tell you to do

  // station parameter
  StationParameter    : ARRAY[1..MAX_STATION] OF ST_STATION_PARAMETER; // wherever, whenever you want. Build it and they will come...

  // station GearInPosCA parameter and data structs
  StationGearParameter: ARRAY[1..MAX_STATION] OF ST_STATION_GEAR_PARAMETER;
  StationGearData     : ARRAY[1..MAX_STATION] OF ST_GEAR_DATA;

  // static position offsets in stations
  PositionOffset      : ARRAY[1..MAX_STATION] OF T_NEST_OFFSET; // added to PosStop[] in XtsStation


  //---------------------------------------------------------------------------
  // XTS
  // XTS TransportUnit
  //  - This is ground control
  //  - handles request for XPU, Group, Mover, StartUp, ReStart
  XtsTransport        : fb_TransportUnit;         // manages members of XTS transport for extern to access

  XtsTransportCtrl    : ST_XTS_TRANSPORT_CTRL;    // control of XTS transport for extern to write
  XtsTransportState   : ST_XTS_TRANSPORT_STATE;   // state   of XTS transport for extern to read


  //---------------------------------------------------------------------------
  // XPU
  // XTS-Utility checks
  // XTS-Utility interfaces for you to use
  Xpu             : fb_XpuCtrl;

  XpuCtrl         : ST_XPU_CTRL;
  XpuState        : ST_XPU_STATE;
  XpuInfo         : ST_XPU_INFO;
  XpuModules      : ARRAY[1..MAX_MODULE] OF Tc3_XTS_Utility.ST_InfoDataView;


  //---------------------------------------------------------------------------
  // Collision avoidance group CA
  //
  // - add mover to group
  // - build group
  // - clear group
  // - whereever you may roam, no on will tread on you
  CaGroup         : FB_CaGroup;                   // cyclic check of CaGroup state and errors; carries methods for handling CaGroup
  CaGroupItf      : I_XtsTransport_CaGroup;       // Interface used by fb_TransportUnit

  // cyclic mapping to MOTION/Objects/CaGroup 
  CaGroupRef      : Tc3_McCoordinatedMotion.AXES_GROUP_REF;

  // Info data from CaGroup FB
  CaGroupInfo     : ST_GROUP_INFO;                // cyclic info about CaGroup for fb_TransportUnit to read
  //---------------------------------------------------------------------------

  //---------------------------------------------------------------------------
  // MC2 encapsulation, CA movement
  Mover           : ARRAY[1..MAX_MOVER] OF fb_MoverCtrl;    // MC and CA methods for mover; cyclic check for individual command on mover

  MoverCtrl       : ARRAY[1..MAX_MOVER] OF ST_MOVER_CTRL;   // control of individual mover for extern to write
  MoverState      : ARRAY[1..MAX_MOVER] OF ST_MOVER_STATE;  // state   of individual mover for extern to read

  MoverItf        : ARRAY[1..MAX_MOVER] OF I_XtsTransport_Mover;  // Interface used by fb_TransportUnit

  LastPosition    : ARRAY[1..MAX_MOVER] OF LREAL;           // on execute of any movement, value is saved here (used by fb_Mover)
  LastGap         : ARRAY[1..MAX_MOVER] OF LREAL;           // on execute of any movement, value is saved here (used by fb_Mover)

  MoverInfo       : ARRAY[1..MAX_MOVER] OF ST_MOVER_INFO;   // cyclic info about mover for extern to read

  MoveData        : ARRAY[1..MAX_MOVER] OF ST_MOVE_DATA;    // dynamic constraints for move commands
  GearData        : ARRAY[1..MAX_MOVER] OF ST_GEAR_DATA;    // dynamic constraints and positions for GearIn/GearInPosCa
  
  // cyclic mapping to MOTION/Axes
  AxisRefMover    : ARRAY[1..MAX_MOVER] OF Tc2_MC2.AXIS_REF;
  //---------------------------------------------------------------------------
END_VAR

// ---- XTS_Parameter_108.TcGVL
//{attribute 'qualified_only'}
VAR_GLOBAL CONSTANT
// HAUD 2025 08 09
//
//    XTS_TRANSPORT_LAYER project
//    
//    MIT License
//    
//    Copyright (c) 2025 HAUD
//    
//    Permission is hereby granted, free of charge, to any person obtaining a copy
//    of this software and associated documentation files (the "Software"), to deal
//    in the Software without restriction, including without limitation the rights
//    to use, copy, modify, merge, publish, distribute, sublicense, and/or sell
//    copies of the Software, and to permit persons to whom the Software is
//    furnished to do so, subject to the following conditions:
//    
//    The above copyright notice and this permission notice shall be included in all
//    copies or substantial portions of the Software.
//    
//    THE SOFTWARE IS PROVIDED "AS IS", WITHOUT WARRANTY OF ANY KIND, EXPRESS OR
//    IMPLIED, INCLUDING BUT NOT LIMITED TO THE WARRANTIES OF MERCHANTABILITY,
//    FITNESS FOR A PARTICULAR PURPOSE AND NONINFRINGEMENT. IN NO EVENT SHALL THE
//    AUTHORS OR COPYRIGHT HOLDERS BE LIABLE FOR ANY CLAIM, DAMAGES OR OTHER
//    LIABILITY, WHETHER IN AN ACTION OF CONTRACT, TORT OR OTHERWISE, ARISING FROM,
//    OUT OF OR IN CONNECTION WITH THE SOFTWARE OR THE USE OR OTHER DEALINGS IN THE
//    SOFTWARE.

  Version             : STRING  := '4.00.11';

  MAX_MOVER           : UINT    := TO_UINT(Tc3_XTS_Utility.TcIoXtsEnvironmentParameterList.MaxXtsMoversPerXpu);
  MAX_MODULE          : UINT    := TO_UINT(Tc3_XTS_Utility.TcIoXtsEnvironmentParameterList.MaxModulesPerPart);
  MAX_PART            : UINT    := TO_UINT(Tc3_XTS_Utility.TcIoXtsEnvironmentParameterList.MaxXtsPartsPerXpu);
  MAX_TRACK           : UINT    := TO_UINT(Tc3_XTS_Utility.TcIoXtsEnvironmentParameterList.MaxXtsTracksPerXpu);
  MAX_GROUP           : UINT    := TO_UINT(Tc3_XTS_Utility.TcIoXtsEnvironmentParameterList.MaxXtsCaGroup);

  MAX_INFO_SERVER     : UINT    := TO_UINT(Tc3_XTS_Utility.TcIoXtsEnvironmentParameterList.MaxXtsInfoServer);
  MAX_INFO_STATION    : UINT    := TO_UINT(Tc3_XTS_Utility.TcIoXtsEnvironmentParameterList.MaxXtsInfoStation);
  MAX_INFO_STOP_POS   : UINT    := TO_UINT(Tc3_XTS_Utility.TcIoXtsEnvironmentParameterList.MaxXtsStopPositionsPerStation);

  MAX_PARAMETER_SET   : UINT    := TO_UINT(Tc3_XTS_Utility.TcIoXtsEnvironmentParameterList.MaxXtsParameterSet);

  MAX_NCT_BASE_UNIT   : UINT    := TO_UINT(Tc3_XTS_Utility.TcIoXtsEnvironmentParameterList.MaxXtsNctBaseUnitInterfaces);

  MAX_STATION         : UINT    := 53;
  MAX_STATION_NEST    : UINT    := TO_UINT(SIZEOF(ST_STATION_STATE.nMask)*8);
  // MAX_LIST_NODES      : UINT    := MAX_MOVER;
  MAX_LIST_NODES      : UINT    := 108; // visualization can not handle access to MAX_MOVER
  MAX_MASTER          : UINT    := 1;
END_VAR

// ---- APPLICATION/_types/Collector/I_ProcessCollector.TcIO
INTERFACE I_ProcessCollector

PROPERTY ActivateStation : DWORD // bit mask for enabling XtsStations in Process
GET
END_GET
END_PROPERTY

METHOD PUBLIC BitDel : T_PROCESS
VAR_INPUT
  inVal   : T_PROCESS;
  bitNo   : DINT;
END_VAR
END_METHOD

METHOD PUBLIC BitGet : BOOL
VAR_INPUT
  inVal   : T_PROCESS;
  bitNo   : DINT;
END_VAR
END_METHOD

METHOD PUBLIC BitSet : T_PROCESS
VAR_INPUT
  inVal   : T_PROCESS;
  bitNo   : DINT;
END_VAR
END_METHOD

METHOD BitsToString : STRING(SIZEOF(T_PROCESS)*8) // T_PROCESS to string
VAR_INPUT
  inVal       : T_PROCESS;
END_VAR
END_METHOD

METHOD Cycle // cyclic call for checking XtsStation state masks and command input from process
END_METHOD

METHOD GetMoverInStation : ST_MOVER_INFO // mover in station info
VAR_INPUT
  nStation            : UINT;   // index of GVL_XTS.StationState[nStation]
END_VAR
END_METHOD

METHOD GetStationState : ST_STATION_STATE
VAR_INPUT
  nStation            : UINT;   // index of GVL_XTS.StationState[nStation]
END_VAR
END_METHOD

METHOD PUBLIC Init : E_PROGRESS // clears all XtsSubstations, then disables all
VAR_INPUT
  Execute     : BOOL;
END_VAR
END_METHOD

PROPERTY MessageLevel : e_MessageType
GET
END_GET
SET
END_SET
END_PROPERTY

PROPERTY ProcessCtrl : reference to st_process_ctrl
GET
END_GET
SET
END_SET
END_PROPERTY

PROPERTY ProcessId : E_INSTANCE
GET
END_GET
SET
END_SET
END_PROPERTY

PROPERTY ProcessState : reference to st_process_state
GET
END_GET
SET
END_SET
END_PROPERTY

PROPERTY QueueMoverIDs : ARRAY[1..SIZEOF(T_PROCESS)*8] OF UINT
GET
END_GET
END_PROPERTY

PROPERTY QueueProcessCount : UINT // sum of all station queues
GET
END_GET
END_PROPERTY

PROPERTY QueueStationCount : ARRAY[1..SIZEOF(T_PROCESS)*8] OF UINT
GET
END_GET
END_PROPERTY

PROPERTY StationCount : UINT
GET
END_GET
END_PROPERTY

PROPERTY StationFirst : uint
GET
END_GET
SET
END_SET
END_PROPERTY

PROPERTY StationLast : uint
GET
END_GET
SET
END_SET
END_PROPERTY

PROPERTY TargetIndex : ARRAY[1..SIZEOF(T_PROCESS)*8] OF USINT
GET
END_GET
SET
END_SET
END_PROPERTY

PROPERTY TargetMask : ARRAY[1..SIZEOF(T_PROCESS)*8] OF BYTE
GET
END_GET
SET
END_SET
END_PROPERTY

METHOD To_T_Process : T_PROCESS // maps (2^nExp)-1 onto T_PROCESS datatype 
VAR_INPUT
  nExp              : BYTE;
END_VAR
END_METHOD

END_INTERFACE

// ---- XTS/CaGroup/I_XtsTransport_CaGroup.TcIO
INTERFACE I_XtsTransport_CaGroup

METHOD AddAll : E_PROGRESS
VAR_INPUT
  Execute     : BOOL;
END_VAR
END_METHOD

METHOD Disable : E_PROGRESS
VAR_INPUT
  Execute     : BOOL;
END_VAR
END_METHOD

METHOD Enable : E_PROGRESS
VAR_INPUT
  Execute     : BOOL;
END_VAR
END_METHOD

METHOD McHaltAll : E_PROGRESS
VAR_INPUT
  Execute       : BOOL;
END_VAR
END_METHOD

METHOD McResetAll : E_PROGRESS
VAR_INPUT
  Execute       : BOOL;
END_VAR
END_METHOD

METHOD RemoveAll : E_PROGRESS
VAR_INPUT
  Execute     : BOOL;
END_VAR
END_METHOD

METHOD Reset : E_PROGRESS
VAR_INPUT
  Execute     : BOOL;
END_VAR
END_METHOD

METHOD Stop : E_PROGRESS
VAR_INPUT
  Execute     : BOOL;
END_VAR
END_METHOD

END_INTERFACE

// ---- XTS/Mover/I_XtsTransport_Mover.TcIO
INTERFACE I_XtsTransport_Mover

METHOD Disable : E_PROGRESS
VAR_INPUT
  Execute             : BOOL;
END_VAR
END_METHOD

METHOD Enable : E_PROGRESS
VAR_INPUT
  Execute             : BOOL;
END_VAR
END_METHOD

METHOD GearIn : E_PROGRESS;
VAR_INPUT
  Execute             : BOOL;
  stMoveData          : ST_MOVE_DATA;
  stGearData          : ST_GEAR_DATA;
END_VAR
END_METHOD

METHOD GearInPosCa : E_PROGRESS
VAR_INPUT
  Execute             : BOOL;
  stMoveData          : ST_MOVE_DATA;
  stGearData          : ST_GEAR_DATA;  
END_VAR
END_METHOD

METHOD GearOut : E_PROGRESS
VAR_INPUT
  Execute             : BOOL;
END_VAR
END_METHOD

METHOD Halt : E_PROGRESS
VAR_INPUT
  Execute             : BOOL;
  stMoveData          : ST_MOVE_DATA;
END_VAR
END_METHOD

METHOD HaltCa : E_PROGRESS
VAR_INPUT
  Execute             : BOOL;
  stMoveData          : ST_MOVE_DATA;
END_VAR
END_METHOD

PROPERTY Master : REFERENCE to AXIS_REF
SET
END_SET
END_PROPERTY

PROPERTY MessageLevel : e_messagetype
SET
END_SET
END_PROPERTY

PROPERTY ModuloTurn : dint
GET
END_GET
END_PROPERTY

METHOD MoveToPos : E_PROGRESS
VAR_INPUT
  Execute             : BOOL;
  stMoveData          : ST_MOVE_DATA;
END_VAR
END_METHOD

METHOD MoveToPosCa : E_PROGRESS
VAR_INPUT
  Execute             : BOOL;
  stMoveData          : ST_MOVE_DATA;
END_VAR
END_METHOD

PROPERTY RailLength : LREAL
GET
END_GET
SET
END_SET
END_PROPERTY

METHOD Reset : E_PROGRESS
VAR_INPUT
  Execute             : BOOL;
END_VAR
END_METHOD

METHOD SendToAbsPosCa : E_PROGRESS
VAR_INPUT
  Execute             : BOOL;
  stMoveData          : ST_MOVE_DATA;
END_VAR
END_METHOD

METHOD SendToModuloPosCa : E_PROGRESS
VAR_INPUT
  Execute             : BOOL;
  stMoveData          : ST_MOVE_DATA;
END_VAR
END_METHOD

METHOD Stop : E_PROGRESS
VAR_INPUT
  Execute             : BOOL;
  stMoveData          : ST_MOVE_DATA;
END_VAR
END_METHOD

END_INTERFACE

// ---- XTS/XtsStation/I_XtsTransport_Station.TcIO
INTERFACE I_XtsTransport_Station

METHOD Init : e_progress
VAR_INPUT
END_VAR
END_METHOD

PROPERTY MessageLevel : e_messagetype
SET
END_SET
END_PROPERTY

PROPERTY TargetWindow : lreal
GET
END_GET
SET
END_SET
END_PROPERTY

END_INTERFACE

// ---- APPLICATION/MAIN_APP.TcPOU
//---------------------------------------------------------------------------------------------------------------
//
//  HAUD 2025.02.24
//
//  - EXAMPLE, change, adapt, use
//  -----------------------------
//  - processes and top level workflow examples
//  - based on fb_Instance for processes
//  - fb_Application as top level control for starting, stopping, restarting etc..
//---------------------------------------------------------------------------------------------------------------
PROGRAM MAIN_APP
VAR
  eInit                       : E_PROGRESS;   // application startup state info

  nProcess                    : uint;
  tonWriteLog                 : Tc2_Standard.TON;
  tWriteLog                   : TIME := T#1S;

  stMsg                       : ST_Message;

  _nBufferOutfeedTarget       : ARRAY[1..2] OF E_INSTANCE;
  _nStnFrst                   : UDINT;

  eMsgState                   : e_message_state;
  eMsgProgress                : E_PROGRESS;
END_VAR

//-----------------------------------------------------------------------------------------------------------------
//-----------------------------------------------------------------------------------------------------------------
// check for MAIN.eInit
//  - wait for fb_TransportUnit to be fully started up
//-----------------------------------------------------------------------------------------------------------------
IF NOT (MAIN.eInit = E_PROGRESS.PROGRESS_DONE) 
THEN 
  eInit                                                     := E_PROGRESS.PROGRESS_INVALID; 
  FOR nProcess := E_INSTANCE.BUFFER_INFEED TO MAX_PROCESS
  DO
    GVL_MSG.MessageLevelProcess[nProcess]                   := GVL_MSG.MessageLevel;
  END_FOR
  //ApplicationMain.MessageLevel                              := GVL_MSG.MessageLevel;

  RETURN; 
END_IF
//-----------------------------------------------------------------------------------------------------------------
// set MAIN_APP message device identification
//-----------------------------------------------------------------------------------------------------------------
stMsg.eDevice                                               := e_Device.Application;
//-----------------------------------------------------------------------------------------------------------------
//-----------------------------------------------------------------------------------------------------------------
//-----------------------------------------------------------------------------------------------------------------
// /assign dataflow
//-----------------------------------------------------------------------------------------------------------------
FOR nProcess := 1 TO MAX_PROCESS
DO
  // identification for inter-process-commands and process ST_MESSAGE.eDevice
  GVL_APPLICATION.ProcessCollector[nProcess].ProcessId      :=    nProcess;

  // linked list for you to use for inter-process-commands (start trigger, exit trigger..)
  GVL_APPLICATION.ItfProcessList[nProcess]                  :=    GVL_APPLICATION.ProcessList[nProcess];

  // give reference of all XtsStations to every process; range of process must be set at startup (see action Init())
  GVL_APPLICATION.ProcessCollector[nProcess].StationCtrl    REF=  GVL_XTS.StationCtrl;
  GVL_APPLICATION.ProcessCollector[nProcess].StationState   REF=  GVL_XTS.StationState;

  GVL_APPLICATION.ProcessCollector[nProcess].MoverInfo      REF=  GVL_XTS.MoverInfo;

  // global interfaces for you to use in your process function blocks
  GVL_APPLICATION.ItfProcessCollector[nProcess]             :=    GVL_APPLICATION.ProcessCollector[nProcess];
END_FOR
//-----------------------------------------------------------------------------------------------------------------
//-----------------------------------------------------------------------------------------------------------------
//-----------------------------------------------------------------------------------------------------------------
//  process instances
//-----------------------------------------------------------------------------------------------------------------
GVL_APPLICATION.TicketControl.ItfList                       :=    GVL_APPLICATION.TicketList;
GVL_APPLICATION.TicketControl.Ctrl                          REF=  GVL_APPLICATION.TicketListControl;
GVL_APPLICATION.TicketControl.State                         REF=  GVL_APPLICATION.TicketListState;
GVL_APPLICATION.TicketControl.NodeDataInput                 REF=  GVL_APPLICATION.TicketListDataInput;
GVL_APPLICATION.TicketControl.NodeDataOutput                REF=  GVL_APPLICATION.TicketListDataOutput;
GVL_APPLICATION.TicketControl.MessageLevel                  :=    GVL_MSG.MessageLevelProcess[e_instance.PROCESS_CONDUCTOR];

GVL_APPLICATION.ProcessConductor.TicketLinkedList           :=    GVL_APPLICATION.TicketList;
GVL_APPLICATION.ProcessConductor.InstanceCtrl               REF=  GVL_APPLICATION.InstanceCtrl;
GVL_APPLICATION.ProcessConductor.InstanceState              REF=  GVL_APPLICATION.InstanceState;
GVL_APPLICATION.ProcessConductor.MessageLevel               :=    GVL_MSG.MessageLevelProcess[e_instance.PROCESS_CONDUCTOR];
GVL_APPLICATION.ProcessConductor.ApplicationVariant         :=    GVL_APPLICATION.AppControl.Variant;

GVL_APPLICATION.BufferInfeed.InstanceCtrl                   REF=  GVL_APPLICATION.InstanceCtrl;
GVL_APPLICATION.BufferInfeed.InstanceState                  REF=  GVL_APPLICATION.InstanceState;
GVL_APPLICATION.BufferInfeed.MessageLevel                   :=    GVL_MSG.MessageLevelProcess[e_instance.BUFFER_INFEED];
                                                            
GVL_APPLICATION.Infeed.InstanceCtrl                         REF=  GVL_APPLICATION.InstanceCtrl;
GVL_APPLICATION.Infeed.InstanceState                        REF=  GVL_APPLICATION.InstanceState;
GVL_APPLICATION.Infeed.MessageLevel                         :=    E_MessageType.eMessageSentient; //GVL_MSG.MessageLevelProcess[e_instance.INFEED];
                                                            
GVL_APPLICATION.BufferOutfeed.InstanceCtrl                  REF=  GVL_APPLICATION.InstanceCtrl;
GVL_APPLICATION.BufferOutfeed.InstanceState                 REF=  GVL_APPLICATION.InstanceState;
GVL_APPLICATION.BufferOutfeed.MessageLevel                  :=    GVL_MSG.MessageLevelProcess[e_instance.BUFFER_OUTFEED];
                                                            
GVL_APPLICATION.Outfeed_R1.InstanceCtrl                     REF=  GVL_APPLICATION.InstanceCtrl;
GVL_APPLICATION.Outfeed_R1.InstanceState                    REF=  GVL_APPLICATION.InstanceState;
GVL_APPLICATION.Outfeed_R1.MessageLevel                     :=    GVL_MSG.MessageLevelProcess[e_instance.OUTFEED_ROBOT_R1];
                                                            
GVL_APPLICATION.Outfeed_R2.InstanceCtrl                     REF=  GVL_APPLICATION.InstanceCtrl;
GVL_APPLICATION.Outfeed_R2.InstanceState                    REF=  GVL_APPLICATION.InstanceState;
GVL_APPLICATION.Outfeed_R2.MessageLevel                     :=    GVL_MSG.MessageLevelProcess[e_instance.OUTFEED_ROBOT_R2];
                                                            
GVL_APPLICATION.SenderFast.InstanceCtrl                     REF=  GVL_APPLICATION.InstanceCtrl;
GVL_APPLICATION.SenderFast.InstanceState                    REF=  GVL_APPLICATION.InstanceState;
GVL_APPLICATION.SenderFast.MessageLevel                     :=    GVL_MSG.MessageLevelProcess[e_instance.SENDER_FAST];
                                                            
GVL_APPLICATION.SenderBufferInfeed.InstanceCtrl             REF=  GVL_APPLICATION.InstanceCtrl;
GVL_APPLICATION.SenderBufferInfeed.InstanceState            REF=  GVL_APPLICATION.InstanceState;
GVL_APPLICATION.SenderBufferInfeed.MessageLevel             :=    GVL_MSG.MessageLevelProcess[e_instance.SENDER_BUFFER_INFEED];
//-----------------------------------------------------------------------------------------------------------------
//-----------------------------------------------------------------------------------------------------------------
//-----------------------------------------------------------------------------------------------------------------
//  main application class
//-----------------------------------------------------------------------------------------------------------------
(*
GVL_APPLICATION.ApplicationMain.Ctrl                        REF=  GVL_APPLICATION.AppControl;
GVL_APPLICATION.ApplicationMain.State                       REF=  GVL_APPLICATION.AppState;
GVL_APPLICATION.ApplicationMain.CollectorInterface          REF=  GVL_APPLICATION.ItfProcessCollector;
GVL_APPLICATION.ApplicationMain.ProcessLinkedLists          REF=  GVL_APPLICATION.ItfProcessList;
GVL_APPLICATION.ApplicationMain.XtsTransportCtrl            REF=  GVL_XTS.XtsTransportCtrl;
GVL_APPLICATION.ApplicationMain.XtsTransportState           REF=  GVL_XTS.XtsTransportState;
GVL_APPLICATION.ApplicationMain.InstanceCtrl                REF=  GVL_APPLICATION.InstanceCtrl;
GVL_APPLICATION.ApplicationMain.InstanceState               REF=  GVL_APPLICATION.InstanceState;
*)
//-----------------------------------------------------------------------------------------------------------------
//-----------------------------------------------------------------------------------------------------------------
//-----------------------------------------------------------------------------------------------------------------
// assign dataflow/
//-----------------------------------------------------------------------------------------------------------------
//-----------------------------------------------------------------------------------------------------------------
//-----------------------------------------------------------------------------------------------------------------
//-----------------------------------------------------------------------------------------------------------------
//  /STARTUP
//
// startup procedure for application
//  - connects processes and XtsStations
//-----------------------------------------------------------------------------------------------------------------
CASE eInit
OF
  E_PROGRESS.PROGRESS_INVALID:                // first cycle startup
    //---------------------------------------------------------------------------------------------------------------
    // first cycle startup
    // - wait for extern to give the command, if we are waiting here MAIN is ready, extern can see that
    //---------------------------------------------------------------------------------------------------------------
    GVL_MSG.ApplicationMessageCtrl.Cmd        := E_MESSAGE_CTRL.MSG_CTRL_NULL;
    eInit                                     := E_PROGRESS.PROGRESS_INIT;

  E_PROGRESS.PROGRESS_INIT:
    //---------------------------------------------------------------------------------------------------------------
    // wait for extern to select valid variant
    //---------------------------------------------------------------------------------------------------------------
      IF (ProcessInitialization(GVL_APPLICATION.AppControl.Variant) = E_PROGRESS.PROGRESS_DONE)
      THEN
        eInit                                 := E_PROGRESS.PROGRESS_BUSY;
      END_IF

  E_PROGRESS.PROGRESS_BUSY:
    //---------------------------------------------------------------------------------------------------------------
    // first cycle startup of all instances
    //---------------------------------------------------------------------------------------------------------------
    GVL_MSG.ApplicationMessageCtrl.Cmd        := E_MESSAGE_CTRL.MSG_CTRL_INIT;

    IF (GVL_MSG.ApplicationMessageState.State = E_MESSAGE_STATE.MSG_STATE_INIT + E_PROGRESS.PROGRESS_DONE)
    THEN
      eInit                                   := E_PROGRESS.PROGRESS_STARTUP;
    END_IF

  E_PROGRESS.PROGRESS_STARTUP:
    IF GVL_MSG.ApplicationMessageData.FileCreated
    THEN
      eInit                                   := E_PROGRESS.PROGRESS_DONE;
      GVL_MSG.ApplicationMessageCtrl.Cmd      := E_MESSAGE_CTRL.MSG_CTRL_NULL;
    END_IF
END_CASE
GVL_APPLICATION.AppState.AppInit              := eInit;
//-----------------------------------------------------------------------------------------------------------------
//-----------------------------------------------------------------------------------------------------------------
// STARTUP/
//-----------------------------------------------------------------------------------------------------------------
//-----------------------------------------------------------------------------------------------------------------
//-----------------------------------------------------------------------------------------------------------------
// /cyclic calls
//-----------------------------------------------------------------------------------------------------------------
//GVL_APPLICATION.ApplicationMain();

GVL_APPLICATION.TicketControl();

GVL_APPLICATION.ProcessConductor();
GVL_APPLICATION.BufferInfeed();
GVL_APPLICATION.Infeed();
GVL_APPLICATION.BufferOutfeed();
GVL_APPLICATION.Outfeed_R1();
GVL_APPLICATION.Outfeed_R2();
GVL_APPLICATION.SenderFast();
GVL_APPLICATION.SenderBufferInfeed();

